KUKA KRL program: MyProgram_204().src

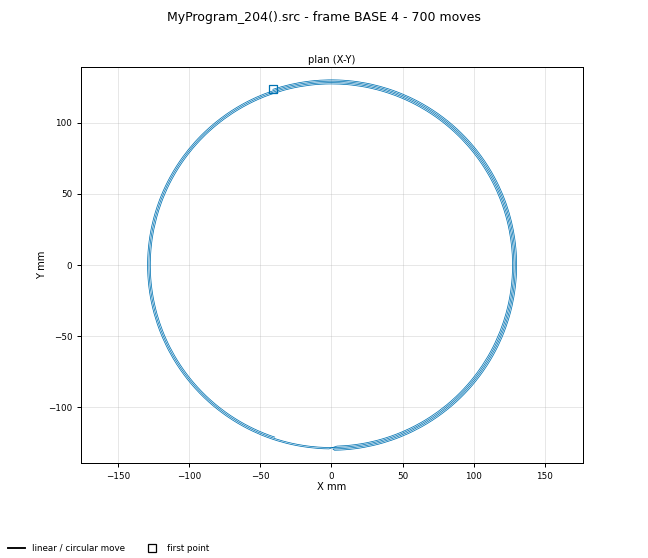
[picture p0: tool path of MyProgram_204().src in frame BASE 4, 700 of 700 moves have a stored position in this frame; points joined in program order, loops and branches not executed]
&ACCESS RVP
&REL 1
&PARAM TEMPLATE = C:\KRC\Roboter\Template\vorgabe
&PARAM EDITMASK = *
DEF MyProgram_204()
; ---- Setting reference (Base) ----
$BASE = BASE_DATA[4]

; --------------------------
; ---- Setting tool (TCP) ----
$TOOL = TOOL_DATA[3]
; --------------------------

$VEL.CP = VEL_APROX_PRINT
Startdeposition()
$VEL.CP = VEL_PRINT
LIN {X -41.1659,Y 123.6241,Z 146,A 104.1591,B 24.9489,C -1.6506,E1 24.9505,E2 342.2401} C_DIS
LIN {X -38.1321,Y 124.5933,Z 146,A 102.7568,B 24.9489,C -1.6522,E1 24.9543,E2 343.6411} C_DIS
LIN {X -35.093,Y 125.4832,Z 146,A 101.3632,B 24.9488,C -1.6536,E1 24.958,E2 345.0335} C_DIS
LIN {X -32.0884,Y 126.285,Z 146,A 100.0013,B 24.9487,C -1.6553,E1 24.9617,E2 346.3934} C_DIS
LIN {X -29.0149,Y 127.0264,Z 146,A 98.5861,B 24.9487,C -1.6553,E1 24.9655,E2 347.8103} C_DIS
LIN {X -25.7092,Y 127.7368,Z 146,A 97.1079,B 24.9485,C -1.6571,E1 24.9696,E2 349.2862} C_DIS
LIN {X -22.6845,Y 128.3085,Z 146,A 95.7157,B 24.9485,C -1.6562,E1 24.9734,E2 350.6819} C_DIS
LIN {X -19.1839,Y 128.8804,Z 146,A 94.052,B 24.9488,C -1.6522,E1 24.978,E2 352.3567} C_DIS
LIN {X -15.434,Y 129.3808,Z 146,A 92.5065,B 24.9484,C -1.6591,E1 24.9823,E2 353.887} C_DIS
LIN {X -12.0776,Y 129.7378,Z 146,A 90.8925,B 24.9488,C -1.6534,E1 24.9868,E2 355.5153} C_DIS
LIN {X -8.0122,Y 130.0517,Z 146,A 89.2662,B 24.9482,C -1.6624,E1 24.9913,E2 357.1208} C_DIS
LIN {X -5.0784,Y 130.1993,Z 146,A 87.9761,B 24.9482,C -1.6629,E1 24.9949,E2 358.4099} C_DIS
LIN {X -2.1677,Y 130.2803,Z 146,A 86.6974,B 24.9482,C -1.6634,E1 24.9984,E2 359.6878} C_DIS
LIN {X 1.1108,Y 130.2942,Z 146,A 85.0901,B 24.9486,C -1.6554,E1 25.003,E2 361.3138} C_DIS
LIN {X 5.0784,Y 130.1993,Z 146,A 83.5047,B 24.9481,C -1.6635,E1 25.0073,E2 362.8796} C_DIS
LIN {X 8.2467,Y 130.0372,Z 146,A 82.0567,B 24.9483,C -1.6609,E1 25.0114,E2 364.3334} C_DIS
LIN {X 11.7081,Y 129.7733,Z 146,A 80.4077,B 24.9487,C -1.6546,E1 25.016,E2 365.9964} C_DIS
LIN {X 15.5086,Y 129.3719,Z 146,A 78.8642,B 24.9483,C -1.6612,E1 25.0203,E2 367.5231} C_DIS
LIN {X 19.1839,Y 128.8804,Z 146,A 77.2629,B 24.9483,C -1.6622,E1 25.0247,E2 369.1206} C_DIS
LIN {X 22.1985,Y 128.3955,Z 146,A 75.9191,B 24.9483,C -1.6617,E1 25.0284,E2 370.4643} C_DIS
LIN {X 24.6619,Y 127.943,Z 146,A 74.7555,B 24.9485,C -1.6581,E1 25.0316,E2 371.635} C_DIS
LIN {X 28.256,Y 127.1998,Z 146,A 73.2021,B 24.9483,C -1.6603,E1 25.0358,E2 373.1811} C_DIS
LIN {X 31.2935,Y 126.4867,Z 146,A 71.8297,B 24.9483,C -1.6595,E1 25.0395,E2 374.5535} C_DIS
LIN {X 34.1145,Y 125.754,Z 146,A 70.5547,B 24.9484,C -1.659,E1 25.043,E2 375.8277} C_DIS
LIN {X 36.8165,Y 124.9886,Z 146,A 69.319,B 24.9484,C -1.6581,E1 25.0463,E2 377.0634} C_DIS
LIN {X 39.9416,Y 124.0254,Z 146,A 67.8799,B 24.9486,C -1.6569,E1 25.0501,E2 378.5028} C_DIS
LIN {X 42.9418,Y 123.0187,Z 146,A 66.4781,B 24.9486,C -1.6552,E1 25.0538,E2 379.906} C_DIS
LIN {X 45.9616,Y 121.9227,Z 146,A 65.0785,B 24.9487,C -1.6545,E1 25.0575,E2 381.3042} C_DIS
LIN {X 49.2138,Y 120.6475,Z 146,A 63.5495,B 24.9487,C -1.6532,E1 25.0615,E2 382.8328} C_DIS
LIN {X 52.4564,Y 119.2749,Z 146,A 61.9925,B 24.9489,C -1.651,E1 25.0655,E2 384.3913} C_DIS
LIN {X 54.9664,Y 118.1368,Z 146,A 60.7346,B 24.9492,C -1.6473,E1 25.0687,E2 385.6549} C_DIS
LIN {X 58.3801,Y 116.4901,Z 146,A 59.1188,B 24.9492,C -1.6477,E1 25.0727,E2 387.2653} C_DIS
LIN {X 61.3057,Y 114.9773,Z 146,A 57.6735,B 24.9492,C -1.6459,E1 25.0763,E2 388.7109} C_DIS
LIN {X 64.563,Y 113.1796,Z 146,A 55.9762,B 24.9496,C -1.6404,E1 25.0804,E2 390.4162} C_DIS
LIN {X 68.0397,Y 111.1243,Z 146,A 54.1884,B 24.9498,C -1.6371,E1 25.0847,E2 392.2062} C_DIS
LIN {X 71.5157,Y 108.9199,Z 146,A 52.38,B 24.95,C -1.6342,E1 25.089,E2 394.0155} C_DIS
LIN {X 74.9755,Y 106.5679,Z 146,A 50.5309,B 24.9502,C -1.6306,E1 25.0932,E2 395.8669} C_DIS
LIN {X 78.6774,Y 103.8649,Z 146,A 48.5505,B 24.9502,C -1.6288,E1 25.0977,E2 397.8444} C_DIS
LIN {X 82.0877,Y 101.1916,Z 146,A 46.6185,B 24.9506,C -1.6238,E1 25.1019,E2 399.7811} C_DIS
LIN {X 85.3172,Y 98.4841,Z 146,A 44.7731,B 24.9508,C -1.6205,E1 25.1058,E2 401.627} C_DIS
LIN {X 88.4903,Y 95.6433,Z 146,A 42.9136,B 24.951,C -1.6173,E1 25.1096,E2 403.4866} C_DIS
LIN {X 91.5168,Y 92.7515,Z 146,A 41.0777,B 24.9512,C -1.6136,E1 25.1133,E2 405.3235} C_DIS
LIN {X 94.4902,Y 89.7205,Z 146,A 39.2228,B 24.9514,C -1.61,E1 25.1169,E2 407.1788} C_DIS
LIN {X 97.316,Y 86.6472,Z 146,A 37.3918,B 24.9517,C -1.6061,E1 25.1204,E2 409.011} C_DIS
LIN {X 100.0901,Y 83.4275,Z 146,A 35.5724,B 24.9517,C -1.6042,E1 25.1236,E2 410.8265} C_DIS
LIN {X 102.7296,Y 80.155,Z 146,A 33.6589,B 24.9523,C -1.5962,E1 25.127,E2 412.7498} C_DIS
LIN {X 105.3588,Y 76.6654,Z 146,A 31.7669,B 24.9525,C -1.5929,E1 25.1301,E2 414.6406} C_DIS
LIN {X 107.8878,Y 73.0632,Z 146,A 29.8878,B 24.9525,C -1.5909,E1 25.1331,E2 416.5153} C_DIS
LIN {X 110.3417,Y 69.3023,Z 146,A 27.9203,B 24.9529,C -1.586,E1 25.1361,E2 418.4845} C_DIS
LIN {X 112.5292,Y 65.691,Z 146,A 26.0522,B 24.9532,C -1.5803,E1 25.1387,E2 420.3563} C_DIS
LIN {X 114.5867,Y 62.0329,Z 146,A 24.2001,B 24.9535,C -1.5748,E1 25.1412,E2 422.2118} C_DIS
LIN {X 116.3208,Y 58.7126,Z 146,A 22.6908,B 24.9534,C -1.5775,E1 25.1431,E2 423.7067} C_DIS
LIN {X 117.7272,Y 55.8387,Z 146,A 21.2514,B 24.9537,C -1.5717,E1 25.1449,E2 425.152} C_DIS
LIN {X 119.2263,Y 52.5651,Z 146,A 19.7299,B 24.9537,C -1.5704,E1 25.1466,E2 426.6685} C_DIS
LIN {X 120.3634,Y 49.9027,Z 146,A 18.4123,B 24.9542,C -1.5642,E1 25.1481,E2 427.9932} C_DIS
LIN {X 122.0195,Y 45.703,Z 146,A 16.484,B 24.9543,C -1.5613,E1 25.15,E2 429.9177} C_DIS
LIN {X 123.1093,Y 42.6806,Z 146,A 15.0884,B 24.9545,C -1.5579,E1 25.1513,E2 431.3134} C_DIS
LIN {X 124.1186,Y 39.6499,Z 146,A 13.6882,B 24.9548,C -1.5539,E1 25.1525,E2 432.7153} C_DIS
LIN {X 125.0483,Y 36.6127,Z 146,A 12.3025,B 24.955,C -1.5501,E1 25.1536,E2 434.1019} C_DIS
LIN {X 125.8983,Y 33.5736,Z 146,A 10.9352,B 24.9552,C -1.5469,E1 25.1546,E2 435.469} C_DIS
LIN {X 126.6698,Y 30.5342,Z 146,A 9.5775,B 24.9554,C -1.5437,E1 25.1556,E2 436.8265} C_DIS
LIN {X 127.3635,Y 27.4977,Z 146,A 8.2079,B 24.9556,C -1.5393,E1 25.1564,E2 438.1984} C_DIS
LIN {X 127.9803,Y 24.4669,Z 146,A 6.8509,B 24.9558,C -1.5351,E1 25.1571,E2 439.5573} C_DIS
LIN {X 128.5213,Y 21.4444,Z 146,A 5.5184,B 24.956,C -1.5317,E1 25.1578,E2 440.89} C_DIS
LIN {X 128.9877,Y 18.4327,Z 146,A 4.1834,B 24.9563,C -1.5277,E1 25.1583,E2 442.2266} C_DIS
LIN {X 129.3808,Y 15.434,Z 146,A 2.8295,B 24.9566,C -1.5221,E1 25.1588,E2 443.5858} C_DIS
LIN {X 129.7733,Y 11.7081,Z 146,A 1.2309,B 24.9568,C -1.5193,E1 25.1592,E2 445.1815} C_DIS
LIN {X 130.0063,Y 8.7481,Z 146,A -0.212,B 24.9574,C -1.5076,E1 25.1595,E2 446.6433} C_DIS
LIN {X 130.1993,Y 5.0784,Z 146,A -1.6641,B 24.9572,C -1.5112,E1 25.1597,E2 448.0784} C_DIS
LIN {X 130.2826,Y 2.0274,Z 146,A -3.0504,B 24.9576,C -1.5043,E1 25.1597,E2 449.4725} C_DIS
LIN {X 130.2851,Y -1.8813,Z 146,A -4.7567,B 24.9579,C -1.4993,E1 25.1597,E2 451.1805} C_DIS
LIN {X 130.1904,Y -5.305,Z 146,A -6.2523,B 24.9581,C -1.4949,E1 25.1597,E2 452.6777} C_DIS
LIN {X 130.0063,Y -8.7481,Z 146,A -7.71,B 24.9582,C -1.493,E1 25.1594,E2 454.1311} C_DIS
LIN {X 129.7229,Y -12.2325,Z 146,A -9.2888,B 24.9586,C -1.4857,E1 25.159,E2 455.7178} C_DIS
LIN {X 129.3524,Y -15.6724,Z 146,A -10.7575,B 24.9588,C -1.4835,E1 25.1585,E2 457.1829} C_DIS
LIN {X 128.8804,Y -19.1839,Z 146,A -12.3029,B 24.959,C -1.479,E1 25.1579,E2 458.7298} C_DIS
LIN {X 128.301,Y -22.7268,Z 146,A -13.9039,B 24.9594,C -1.4727,E1 25.1572,E2 460.3365} C_DIS
LIN {X 127.6814,Y -25.9814,Z 146,A -15.323,B 24.9595,C -1.4699,E1 25.1564,E2 461.7538} C_DIS
LIN {X 127.0264,Y -29.0149,Z 146,A -16.6968,B 24.9598,C -1.465,E1 25.1556,E2 463.1313} C_DIS
LIN {X 126.2312,Y -32.3004,Z 146,A -18.1777,B 24.96,C -1.4604,E1 25.1546,E2 464.6143} C_DIS
LIN {X 125.3725,Y -35.489,Z 146,A -19.6315,B 24.9603,C -1.4556,E1 25.1535,E2 466.071} C_DIS
LIN {X 124.4556,Y -38.5819,Z 146,A -21.0351,B 24.9605,C -1.4518,E1 25.1524,E2 467.4756} C_DIS
LIN {X 123.4403,Y -41.7177,Z 146,A -22.4398,B 24.9606,C -1.4496,E1 25.1511,E2 468.8776} C_DIS
LIN {X 122.5066,Y -44.3814,Z 146,A -23.7072,B 24.9609,C -1.4442,E1 25.1499,E2 470.1505} C_DIS
LIN {X 121.2828,Y -47.6258,Z 146,A -25.1893,B 24.9611,C -1.4417,E1 25.1485,E2 471.6303} C_DIS
LIN {X 120.0731,Y -50.5978,Z 146,A -26.6249,B 24.9614,C -1.436,E1 25.1469,E2 473.0716} C_DIS
LIN {X 118.7918,Y -53.5364,Z 146,A -28.0489,B 24.9617,C -1.4308,E1 25.1453,E2 474.5} C_DIS
LIN {X 117.472,Y -56.3728,Z 146,A -29.3837,B 24.9617,C -1.4288,E1 25.1437,E2 475.8324} C_DIS
LIN {X 115.9248,Y -59.4905,Z 146,A -31.0338,B 24.9624,C -1.4177,E1 25.1416,E2 477.4999} C_DIS
LIN {X 113.7905,Y -63.4816,Z 146,A -33.0095,B 24.9626,C -1.4124,E1 25.139,E2 479.4776} C_DIS
LIN {X 111.5808,Y -67.2886,Z 146,A -34.8948,B 24.9628,C -1.4094,E1 25.1363,E2 481.3603} C_DIS
LIN {X 109.288,Y -70.9517,Z 146,A -36.7607,B 24.963,C -1.4057,E1 25.1335,E2 483.2254} C_DIS
LIN {X 106.9636,Y -74.4097,Z 146,A -38.5852,B 24.9632,C -1.4009,E1 25.1306,E2 485.0524} C_DIS
LIN {X 104.5125,Y -77.8148,Z 146,A -40.4188,B 24.9635,C -1.3964,E1 25.1276,E2 486.8879} C_DIS
LIN {X 101.9488,Y -81.1445,Z 146,A -42.2562,B 24.9637,C -1.3918,E1 25.1244,E2 488.7273} C_DIS
LIN {X 99.2765,Y -84.393,Z 146,A -44.096,B 24.9639,C -1.3874,E1 25.1211,E2 490.5691} C_DIS
LIN {X 96.6485,Y -87.3906,Z 146,A -45.8895,B 24.9643,C -1.3807,E1 25.1178,E2 492.3705} C_DIS
LIN {X 93.6143,Y -90.6331,Z 146,A -47.775,B 24.9643,C -1.3793,E1 25.1142,E2 494.2511} C_DIS
LIN {X 90.6331,Y -93.6143,Z 146,A -49.6264,B 24.9646,C -1.3748,E1 25.1105,E2 496.1052} C_DIS
LIN {X 87.606,Y -96.453,Z 146,A -51.4433,B 24.9648,C -1.3708,E1 25.1067,E2 497.9241} C_DIS
LIN {X 84.5251,Y -99.1642,Z 146,A -53.2748,B 24.9651,C -1.3652,E1 25.1029,E2 499.7618} C_DIS
LIN {X 81.1445,Y -101.9488,Z 146,A -55.1532,B 24.9651,C -1.3633,E1 25.0988,E2 501.6374} C_DIS
LIN {X 77.8179,Y -104.5102,Z 146,A -56.9762,B 24.9653,C -1.3605,E1 25.0947,E2 503.4603} C_DIS
LIN {X 74.5281,Y -106.8812,Z 146,A -58.7931,B 24.9656,C -1.355,E1 25.0906,E2 505.284} C_DIS
LIN {X 70.9517,Y -109.288,Z 146,A -60.6507,B 24.9657,C -1.3532,E1 25.0863,E2 507.1397} C_DIS
LIN {X 67.1938,Y -111.6381,Z 146,A -62.622,B 24.966,C -1.3483,E1 25.0816,E2 509.1164} C_DIS
LIN {X 63.4816,Y -113.7905,Z 146,A -64.4818,B 24.966,C -1.3462,E1 25.0771,E2 510.9755} C_DIS
LIN {X 59.8462,Y -115.7437,Z 146,A -66.2101,B 24.966,C -1.3476,E1 25.0728,E2 512.6957} C_DIS
LIN {X 57.3676,Y -116.9896,Z 146,A -67.4374,B 24.9661,C -1.3452,E1 25.0697,E2 513.9254} C_DIS
LIN {X 53.9453,Y -118.6089,Z 146,A -69.0822,B 24.9661,C -1.3435,E1 25.0656,E2 515.5699} C_DIS
LIN {X 51.2764,Y -119.7851,Z 146,A -70.3402,B 24.9662,C -1.3429,E1 25.0623,E2 516.8264} C_DIS
LIN {X 48.2339,Y -121.0425,Z 146,A -71.7953,B 24.9663,C -1.3404,E1 25.0586,E2 518.2841} C_DIS
LIN {X 45.3511,Y -122.1513,Z 146,A -73.1766,B 24.9665,C -1.3373,E1 25.055,E2 519.6697} C_DIS
LIN {X 42.2564,Y -123.2564,Z 146,A -74.5919,B 24.9665,C -1.337,E1 25.0512,E2 521.083} C_DIS
LIN {X 39.2006,Y -124.2621,Z 146,A -76.023,B 24.9667,C -1.3343,E1 25.0474,E2 522.5176} C_DIS
LIN {X 36.3649,Y -125.1208,Z 146,A -77.3394,B 24.9667,C -1.3321,E1 25.0439,E2 523.8369} C_DIS
LIN {X 32.9264,Y -126.0709,Z 146,A -78.9998,B 24.9671,C -1.3257,E1 25.0394,E2 525.5101} C_DIS
LIN {X 29.1313,Y -126.9998,Z 146,A -80.599,B 24.9669,C -1.3301,E1 25.0351,E2 527.0963} C_DIS
LIN {X 25.9814,Y -127.6814,Z 146,A -81.9862,B 24.9669,C -1.3304,E1 25.0313,E2 528.4812} C_DIS
LIN {X 22.9743,Y -128.2567,Z 146,A -83.332,B 24.9669,C -1.3293,E1 25.0276,E2 529.8281} C_DIS
LIN {X 19.937,Y -128.7638,Z 146,A -84.7073,B 24.967,C -1.3272,E1 25.0238,E2 531.2071} C_DIS
LIN {X 16.5645,Y -129.2415,Z 146,A -86.2017,B 24.967,C -1.3263,E1 25.0196,E2 532.7022} C_DIS
LIN {X 13.1951,Y -129.6305,Z 146,A -87.658,B 24.967,C -1.3272,E1 25.0156,E2 534.1554} C_DIS
LIN {X 9.6067,Y -129.9437,Z 146,A -89.2621,B 24.967,C -1.3254,E1 25.0111,E2 535.7628} C_DIS
LIN {X 6.2428,Y -130.149,Z 146,A -90.8764,B 24.9675,C -1.3181,E1 25.0066,E2 537.394} C_DIS
LIN {X 2.1677,Y -130.2803,Z 146,A -92.503,B 24.9671,C -1.326,E1 25.0021,E2 539.0016} C_DIS
LIN {X 2.1677,Y -130.2803,Z 146,A -92.503,B 24.9671,C -1.326,E1 25.0021,E2 539.0016} C_DIS
Enddeposition()
LIN {X 0.9239,Y -129.3368,Z 146,A -93.0172,B 24.1837,C -1.1824,E1 24.2108,E2 539.7577} C_DIS
Startdeposition()
$VEL.CP = VEL_PRINT
LIN {X 4.2044,Y -129.2745,Z 146,A -90.6178,B 24.1815,C -1.2293,E1 24.2178,E2 537.2441} C_DIS
LIN {X 8.0458,Y -129.0909,Z 146,A -88.9904,B 24.1816,C -1.2262,E1 24.2223,E2 535.6249} C_DIS
LIN {X 12.9463,Y -128.693,Z 146,A -86.7775,B 24.1815,C -1.2291,E1 24.2285,E2 533.4063} C_DIS
LIN {X 16.7077,Y -128.2576,Z 146,A -84.5287,B 24.18,C -1.2589,E1 24.2349,E2 531.0866} C_DIS
LIN {X 21.7471,Y -127.5007,Z 146,A -83.0315,B 24.1818,C -1.2223,E1 24.2388,E2 529.6803} C_DIS
LIN {X 24.389,Y -127.0209,Z 146,A -81.7505,B 24.1815,C -1.2279,E1 24.2423,E2 528.3873} C_DIS
LIN {X 27.9389,Y -126.2892,Z 146,A -80.0921,B 24.1813,C -1.232,E1 24.2469,E2 526.7211} C_DIS
LIN {X 31.6964,Y -125.3972,Z 146,A -78.4252,B 24.1813,C -1.2315,E1 24.2514,E2 525.0579} C_DIS
LIN {X 35.0406,Y -124.5042,Z 146,A -76.8855,B 24.1813,C -1.2335,E1 24.2555,E2 523.5159} C_DIS
LIN {X 39.6598,Y -123.1109,Z 146,A -74.8628,B 24.1814,C -1.2302,E1 24.2609,E2 521.505} C_DIS
LIN {X 42.3734,Y -122.203,Z 146,A -73.4996,B 24.1811,C -1.2366,E1 24.2645,E2 520.1288} C_DIS
LIN {X 45.6538,Y -121.0161,Z 146,A -71.9964,B 24.1811,C -1.2366,E1 24.2685,E2 518.6291} C_DIS
LIN {X 48.6388,Y -119.8475,Z 146,A -70.5355,B 24.1809,C -1.2407,E1 24.2723,E2 517.1616} C_DIS
LIN {X 53.521,Y -117.7505,Z 146,A -68.2298,B 24.1809,C -1.2418,E1 24.2782,E2 514.8591} C_DIS
LIN {X 56.6438,Y -116.2796,Z 146,A -66.5962,B 24.1805,C -1.2496,E1 24.2823,E2 513.2109} C_DIS
LIN {X 64.9061,Y -111.8783,Z 146,A -62.4943,B 24.1802,C -1.2545,E1 24.2924,E2 509.1093} C_DIS
LIN {X 70.1129,Y -108.6914,Z 146,A -59.8427,B 24.1802,C -1.2569,E1 24.2987,E2 506.4605} C_DIS
LIN {X 73.18,Y -106.65,Z 146,A -58.1557,B 24.1798,C -1.2631,E1 24.3026,E2 504.7644} C_DIS
LIN {X 76.8503,Y -104.037,Z 146,A -56.1353,B 24.1796,C -1.2685,E1 24.3072,E2 502.7382} C_DIS
LIN {X 80.3501,Y -101.3581,Z 146,A -54.1965,B 24.1794,C -1.2721,E1 24.3114,E2 500.7982} C_DIS
LIN {X 83.8862,Y -98.4513,Z 146,A -52.2016,B 24.1792,C -1.275,E1 24.3157,E2 498.8041} C_DIS
LIN {X 87.2035,Y -95.5261,Z 146,A -49.7022,B 24.1776,C -1.3078,E1 24.321,E2 496.2355} C_DIS
LIN {X 90.7593,Y -92.1532,Z 146,A -48.3526,B 24.1795,C -1.2703,E1 24.3235,E2 494.9828} C_DIS
LIN {X 92.8609,Y -90.0356,Z 146,A -46.81,B 24.1787,C -1.285,E1 24.3266,E2 493.4112} C_DIS
LIN {X 95.6119,Y -87.109,Z 146,A -44.9804,B 24.1784,C -1.2922,E1 24.3301,E2 491.5726} C_DIS
LIN {X 98.4763,Y -83.8568,Z 146,A -43.0739,B 24.1782,C -1.2965,E1 24.3336,E2 489.6645} C_DIS
LIN {X 101.4916,Y -80.1818,Z 146,A -41.0186,B 24.178,C -1.2996,E1 24.3372,E2 487.6117} C_DIS
LIN {X 104.0224,Y -76.8701,Z 146,A -39.1282,B 24.1776,C -1.3069,E1 24.3403,E2 485.7128} C_DIS
LIN {X 106.9996,Y -72.6683,Z 146,A -36.1292,B 24.1753,C -1.3512,E1 24.3452,E2 482.6216} C_DIS
LIN {X 110.2998,Y -67.5537,Z 146,A -34.2932,B 24.1773,C -1.3136,E1 24.3478,E2 480.8865} C_DIS
LIN {X 112.8544,Y -63.1939,Z 146,A -32.051,B 24.1769,C -1.3204,E1 24.3509,E2 478.6399} C_DIS
LIN {X 114.62,Y -59.9279,Z 146,A -30.468,B 24.1769,C -1.3221,E1 24.353,E2 477.0613} C_DIS
LIN {X 116.1533,Y -56.8998,Z 146,A -28.9363,B 24.1765,C -1.3281,E1 24.3549,E2 475.5235} C_DIS
LIN {X 118.4291,Y -52.0014,Z 146,A -26.6306,B 24.1765,C -1.3309,E1 24.3576,E2 473.2241} C_DIS
LIN {X 119.4601,Y -49.5826,Z 146,A -25.4584,B 24.1762,C -1.3349,E1 24.3588,E2 472.0488} C_DIS
LIN {X 120.616,Y -46.6999,Z 146,A -24.0694,B 24.1759,C -1.3399,E1 24.3603,E2 470.6557} C_DIS
LIN {X 121.8745,Y -43.3132,Z 146,A -22.1514,B 24.1748,C -1.3617,E1 24.3621,E2 468.696} C_DIS
LIN {X 122.971,Y -40.0975,Z 146,A -21.0036,B 24.1755,C -1.3476,E1 24.3631,E2 467.5891} C_DIS
LIN {X 124.0699,Y -36.5487,Z 146,A -19.4234,B 24.1755,C -1.3495,E1 24.3644,E2 466.0136} C_DIS
LIN {X 124.9718,Y -33.3341,Z 146,A -17.8718,B 24.175,C -1.358,E1 24.3655,E2 464.4505} C_DIS
LIN {X 125.8855,Y -29.7043,Z 146,A -16.1834,B 24.1746,C -1.365,E1 24.3666,E2 462.7554} C_DIS
LIN {X 126.7224,Y -25.8954,Z 146,A -14.5182,B 24.1745,C -1.3673,E1 24.3676,E2 461.0945} C_DIS
LIN {X 127.3956,Y -22.3539,Z 146,A -12.8758,B 24.1741,C -1.3749,E1 24.3684,E2 459.4437} C_DIS
LIN {X 128.2631,Y -16.6661,Z 146,A -9.9027,B 24.1724,C -1.4057,E1 24.3696,E2 456.4141} C_DIS
LIN {X 128.7367,Y -12.4917,Z 146,A -8.6813,B 24.1739,C -1.378,E1 24.3699,E2 455.2673} C_DIS
LIN {X 129.1577,Y -6.9019,Z 146,A -5.9341,B 24.1727,C -1.4,E1 24.3705,E2 452.4836} C_DIS
LIN {X 129.3221,Y -2.2358,Z 146,A -4.0351,B 24.1729,C -1.3979,E1 24.3705,E2 450.6016} C_DIS
LIN {X 129.3232,Y 2.17,Z 146,A -1.5858,B 24.1711,C -1.4305,E1 24.3705,E2 448.0881} C_DIS
LIN {X 129.1818,Y 6.4224,Z 146,A -0.2608,B 24.1723,C -1.4071,E1 24.3704,E2 446.8281} C_DIS
LIN {X 128.8041,Y 11.7869,Z 146,A 2.2966,B 24.1714,C -1.424,E1 24.3698,E2 444.2454} C_DIS
LIN {X 128.3691,Y 15.837,Z 146,A 4.6153,B 24.1696,C -1.457,E1 24.369,E2 441.8609} C_DIS
LIN {X 127.6433,Y 20.8922,Z 146,A 6.1983,B 24.1712,C -1.4284,E1 24.3683,E2 440.3569} C_DIS
LIN {X 126.9954,Y 24.5227,Z 146,A 7.8199,B 24.1709,C -1.433,E1 24.3675,E2 438.734} C_DIS
LIN {X 126.1682,Y 28.4747,Z 146,A 9.6145,B 24.1706,C -1.4389,E1 24.3664,E2 436.9358} C_DIS
LIN {X 125.37,Y 31.8035,Z 146,A 11.0633,B 24.1706,C -1.4401,E1 24.3655,E2 435.4927} C_DIS
LIN {X 124.5497,Y 34.8778,Z 146,A 12.4941,B 24.1702,C -1.4456,E1 24.3644,E2 434.0571} C_DIS
LIN {X 123.4683,Y 38.5381,Z 146,A 14.3531,B 24.1694,C -1.4596,E1 24.3629,E2 432.1753} C_DIS
LIN {X 122.19,Y 42.4108,Z 146,A 15.9591,B 24.1697,C -1.4546,E1 24.3615,E2 430.5906} C_DIS
LIN {X 121.0601,Y 45.5363,Z 146,A 17.4246,B 24.1695,C -1.4587,E1 24.36,E2 429.1237} C_DIS
LIN {X 119.9067,Y 48.4921,Z 146,A 18.8661,B 24.1691,C -1.4647,E1 24.3585,E2 427.6758} C_DIS
LIN {X 118.1026,Y 52.7336,Z 146,A 20.8906,B 24.1688,C -1.4698,E1 24.3563,E2 425.6506} C_DIS
LIN {X 116.6258,Y 55.9241,Z 146,A 22.3968,B 24.1688,C -1.4716,E1 24.3545,E2 424.1484} C_DIS
LIN {X 115.0671,Y 59.066,Z 146,A 23.947,B 24.1685,C -1.4758,E1 24.3525,E2 422.5965} C_DIS
LIN {X 113.2636,Y 62.4577,Z 146,A 25.7619,B 24.1679,C -1.4864,E1 24.3501,E2 420.7658} C_DIS
LIN {X 111.3295,Y 65.8441,Z 146,A 27.4692,B 24.1677,C -1.49,E1 24.3477,E2 419.0587} C_DIS
LIN {X 108.9731,Y 69.6736,Z 146,A 29.2932,B 24.1679,C -1.4867,E1 24.345,E2 417.2524} C_DIS
LIN {X 106.8718,Y 72.8569,Z 146,A 31.0848,B 24.1673,C -1.4963,E1 24.3422,E2 415.4466} C_DIS
LIN {X 104.4728,Y 76.257,Z 146,A 32.9722,B 24.1669,C -1.5033,E1 24.3391,E2 413.5517} C_DIS
LIN {X 101.074,Y 80.7071,Z 146,A 35.1506,B 24.1675,C -1.4939,E1 24.3355,E2 411.4069} C_DIS
LIN {X 99.1815,Y 83.0217,Z 146,A 36.7336,B 24.1665,C -1.5103,E1 24.3326,E2 409.7916} C_DIS
LIN {X 96.1606,Y 86.5029,Z 146,A 39.5696,B 24.1638,C -1.556,E1 24.3271,E2 406.8575} C_DIS
LIN {X 91.85,Y 91.0667,Z 146,A 41.4539,B 24.1662,C -1.5159,E1 24.3237,E2 405.079} C_DIS
LIN {X 88.7788,Y 94.0631,Z 146,A 43.4094,B 24.1658,C -1.5228,E1 24.3197,E2 403.1153} C_DIS
LIN {X 85.4833,Y 97.0681,Z 146,A 45.3703,B 24.1656,C -1.526,E1 24.3156,E2 401.1546} C_DIS
LIN {X 81.609,Y 100.3473,Z 146,A 47.3329,B 24.1662,C -1.5159,E1 24.3115,E2 399.2244} C_DIS
LIN {X 78.0777,Y 103.1186,Z 146,A 49.6182,B 24.1651,C -1.5346,E1 24.3064,E2 396.9024} C_DIS
LIN {X 74.4187,Y 105.7896,Z 146,A 51.5752,B 24.165,C -1.5356,E1 24.3019,E2 394.9502} C_DIS
LIN {X 70.9411,Y 108.1525,Z 146,A 53.4624,B 24.1647,C -1.5399,E1 24.2975,E2 393.059} C_DIS
LIN {X 67.0886,Y 110.5834,Z 146,A 55.4658,B 24.1646,C -1.5423,E1 24.2928,E2 391.0562} C_DIS
LIN {X 63.4058,Y 112.7353,Z 146,A 57.3529,B 24.1644,C -1.545,E1 24.2882,E2 389.1685} C_DIS
LIN {X 59.5391,Y 114.8242,Z 146,A 59.1768,B 24.1646,C -1.5415,E1 24.2837,E2 387.3585} C_DIS
LIN {X 56.593,Y 116.3047,Z 146,A 60.7468,B 24.1642,C -1.5488,E1 24.2798,E2 385.7751} C_DIS
LIN {X 53.0349,Y 117.9679,Z 146,A 62.4099,B 24.1643,C -1.5471,E1 24.2756,E2 384.1205} C_DIS
LIN {X 49.5936,Y 119.4555,Z 146,A 64.0262,B 24.1643,C -1.5467,E1 24.2714,E2 382.5092} C_DIS
LIN {X 46.6078,Y 120.6518,Z 146,A 65.4667,B 24.1642,C -1.5489,E1 24.2677,E2 381.0665} C_DIS
LIN {X 43.0618,Y 121.9643,Z 146,A 67.2656,B 24.1637,C -1.5566,E1 24.2629,E2 379.2528} C_DIS
LIN {X 39.0091,Y 123.3188,Z 146,A 69.018,B 24.1641,C -1.5512,E1 24.2583,E2 377.5168} C_DIS
LIN {X 35.3983,Y 124.4042,Z 146,A 70.7735,B 24.1637,C -1.5567,E1 24.2536,E2 375.7512} C_DIS
LIN {X 31.7622,Y 125.3805,Z 146,A 72.3687,B 24.1639,C -1.5542,E1 24.2493,E2 374.1647} C_DIS
LIN {X 28.7121,Y 126.114,Z 146,A 73.7517,B 24.1639,C -1.5546,E1 24.2455,E2 372.7825} C_DIS
LIN {X 25.5775,Y 126.7871,Z 146,A 75.1911,B 24.1638,C -1.5562,E1 24.2416,E2 371.3411} C_DIS
LIN {X 21.5757,Y 127.5293,Z 146,A 77.3254,B 24.1627,C -1.5732,E1 24.2356,E2 369.1679} C_DIS
LIN {X 18.1742,Y 128.058,Z 146,A 78.9804,B 24.1623,C -1.58,E1 24.231,E2 367.4977} C_DIS
LIN {X 14.0715,Y 128.5737,Z 146,A 80.3449,B 24.1637,C -1.5574,E1 24.2274,E2 366.1893} C_DIS
LIN {X 9.1632,Y 129.0166,Z 146,A 82.4892,B 24.1637,C -1.5557,E1 24.2214,E2 364.0503} C_DIS
LIN {X 6.1891,Y 129.1935,Z 146,A 84.2824,B 24.1624,C -1.5787,E1 24.2163,E2 362.2016} C_DIS
LIN {X 2.2488,Y 129.3219,Z 146,A 85.5423,B 24.1638,C -1.5549,E1 24.2129,E2 361.0002} C_DIS
LIN {X -1.1826,Y 129.3368,Z 146,A 87.6507,B 24.1621,C -1.5831,E1 24.2068,E2 358.8229} C_DIS
LIN {X -5.6719,Y 129.2183,Z 146,A 89.0697,B 24.1638,C -1.5548,E1 24.2031,E2 357.4726} C_DIS
LIN {X -10.4326,Y 128.9207,Z 146,A 91.3757,B 24.1633,C -1.5632,E1 24.1966,E2 355.1452} C_DIS
LIN {X -14.4334,Y 128.5348,Z 146,A 93.4781,B 24.1624,C -1.5777,E1 24.1906,E2 353.0059} C_DIS
LIN {X -18.4741,Y 128.0152,Z 146,A 94.6681,B 24.1643,C -1.5471,E1 24.1876,E2 351.8898} C_DIS
LIN {X -21.3457,Y 127.5676,Z 146,A 96.0606,B 24.1641,C -1.5512,E1 24.1837,E2 350.486} C_DIS
LIN {X -24.6883,Y 126.9637,Z 146,A 97.7247,B 24.1637,C -1.5576,E1 24.1791,E2 348.8044} C_DIS
LIN {X -28.795,Y 126.0951,Z 146,A 99.456,B 24.1641,C -1.5499,E1 24.1744,E2 347.0898} C_DIS
LIN {X -32.5621,Y 125.1775,Z 146,A 101.2988,B 24.1639,C -1.5541,E1 24.1694,E2 345.234} C_DIS
LIN {X -36.2023,Y 124.1713,Z 146,A 102.98,B 24.1639,C -1.5527,E1 24.1648,E2 343.5533} C_DIS
LIN {X -39.6345,Y 123.119,Z 146,A 104.4461,B 24.1644,C -1.545,E1 24.161,E2 342.1034} C_DIS
LIN {X -47.1522,Y 120.4402,Z 146,A 108.0019,B 24.1647,C -1.5413,E1 24.1517,E2 338.5492} C_DIS
LIN {X -52.6198,Y 118.1536,Z 146,A 110.3757,B 24.1656,C -1.5257,E1 24.1457,E2 336.2079} C_DIS
LIN {X -56.0134,Y 116.5831,Z 146,A 112.2625,B 24.1651,C -1.5339,E1 24.1408,E2 334.2962} C_DIS
LIN {X -59.0106,Y 115.0953,Z 146,A 113.8105,B 24.1651,C -1.5345,E1 24.1369,E2 332.7424} C_DIS
LIN {X -62.8395,Y 113.0522,Z 146,A 115.808,B 24.1651,C -1.5347,E1 24.132,E2 330.7385} C_DIS
LIN {X -66.6481,Y 110.8499,Z 146,A 117.7933,B 24.1651,C -1.5328,E1 24.1272,E2 328.7516} C_DIS
LIN {X -70.4343,Y 108.483,Z 146,A 120.1018,B 24.1645,C -1.5444,E1 24.1217,E2 326.4069} C_DIS
LIN {X -73.7242,Y 106.2748,Z 146,A 122.1725,B 24.1638,C -1.5556,E1 24.1169,E2 324.3014} C_DIS
LIN {X -78.1894,Y 103.0344,Z 146,A 123.7093,B 24.1666,C -1.5083,E1 24.1137,E2 322.875} C_DIS
LIN {X -81.9997,Y 100.0281,Z 146,A 126.1808,B 24.166,C -1.5184,E1 24.1083,E2 320.3692} C_DIS
LIN {X -85.5473,Y 97.0114,Z 146,A 128.212,B 24.1664,C -1.5122,E1 24.104,E2 318.3449} C_DIS
LIN {X -88.9697,Y 93.883,Z 146,A 130.5078,B 24.166,C -1.5185,E1 24.0992,E2 316.0239} C_DIS
LIN {X -91.4109,Y 91.508,Z 146,A 132.0358,B 24.1662,C -1.5157,E1 24.0962,E2 314.4961} C_DIS
LIN {X -93.8238,Y 89.0325,Z 146,A 133.0862,B 24.1677,C -1.4898,E1 24.0943,E2 313.5046} C_DIS
LIN {X -95.9392,Y 86.7483,Z 146,A 134.675,B 24.1673,C -1.4959,E1 24.0913,E2 311.8935} C_DIS
LIN {X -100.6523,Y 81.2321,Z 146,A 137.74,B 24.1682,C -1.4806,E1 24.0858,E2 308.8514} C_DIS
LIN {X -104.3902,Y 76.3694,Z 146,A 140.5807,B 24.1683,C -1.4788,E1 24.081,E2 306.001} C_DIS
LIN {X -106.7035,Y 73.1021,Z 146,A 142.417,B 24.1684,C -1.4767,E1 24.078,E2 304.1604} C_DIS
LIN {X -109.0948,Y 69.4835,Z 146,A 144.4029,B 24.1686,C -1.4742,E1 24.075,E2 302.1704} C_DIS
LIN {X -111.3739,Y 65.7684,Z 146,A 146.3566,B 24.1688,C -1.4697,E1 24.0722,E2 300.2174} C_DIS
LIN {X -113.6346,Y 61.78,Z 146,A 148.3805,B 24.1692,C -1.4634,E1 24.0695,E2 298.198} C_DIS
LIN {X -115.3403,Y 58.5294,Z 146,A 149.8692,B 24.1698,C -1.4523,E1 24.0676,E2 296.7281} C_DIS
LIN {X -116.7979,Y 55.5639,Z 146,A 151.4145,B 24.1698,C -1.4515,E1 24.0657,E2 295.176} C_DIS
LIN {X -118.3871,Y 52.0977,Z 146,A 153.1821,B 24.17,C -1.4499,E1 24.0637,E2 293.4024} C_DIS
LIN {X -120.2037,Y 47.7553,Z 146,A 155.1596,B 24.1706,C -1.4386,E1 24.0616,E2 291.4414} C_DIS
LIN {X -121.3081,Y 44.8742,Z 146,A 157.1033,B 24.1694,C -1.4605,E1 24.0597,E2 289.4323} C_DIS
LIN {X -122.7332,Y 40.8124,Z 146,A 158.1312,B 24.1719,C -1.4147,E1 24.0589,E2 288.511} C_DIS
LIN {X -123.9982,Y 36.7936,Z 146,A 160.2194,B 24.1717,C -1.4187,E1 24.0571,E2 286.4004} C_DIS
LIN {X -125.0479,Y 33.0487,Z 146,A 162.1282,B 24.1716,C -1.4216,E1 24.0556,E2 284.4731} C_DIS
LIN {X -126.3127,Y 27.8299,Z 146,A 164.5779,B 24.1718,C -1.4171,E1 24.0541,E2 282.0195} C_DIS
LIN {X -127.048,Y 24.2471,Z 146,A 166.1364,B 24.1722,C -1.4091,E1 24.0532,E2 280.4711} C_DIS
LIN {X -127.7251,Y 20.3912,Z 146,A 167.9716,B 24.1723,C -1.4079,E1 24.0524,E2 278.6274} C_DIS
LIN {X -128.2633,Y 16.6644,Z 146,A 169.6083,B 24.1727,C -1.4011,E1 24.0518,E2 276.9973} C_DIS
LIN {X -128.7404,Y 12.4535,Z 146,A 171.447,B 24.1731,C -1.3932,E1 24.0512,E2 275.1665} C_DIS
LIN {X -129.0447,Y 8.7784,Z 146,A 173.2366,B 24.1731,C -1.3949,E1 24.0509,E2 273.3617} C_DIS
LIN {X -129.258,Y 4.6588,Z 146,A 175.0395,B 24.1734,C -1.3878,E1 24.0507,E2 271.5649} C_DIS
LIN {X -129.344,Y 0.3403,Z 146,A 177.0307,B 24.1735,C -1.3851,E1 24.0507,E2 269.568} C_DIS
LIN {X -129.2872,Y -3.7469,Z 146,A 178.6919,B 24.1742,C -1.3724,E1 24.0507,E2 267.9275} C_DIS
LIN {X -129.108,Y -7.7669,Z 146,A -179.505,B 24.1745,C -1.3676,E1 24.051,E2 266.1251} C_DIS
LIN {X -128.8318,Y -11.4843,Z 146,A -177.7439,B 24.1745,C -1.3672,E1 24.0514,E2 264.3539} C_DIS
LIN {X -128.4217,Y -15.3954,Z 146,A -176.1034,B 24.175,C -1.357,E1 24.0519,E2 262.7283} C_DIS
LIN {X -127.897,Y -19.281,Z 146,A -174.2729,B 24.1751,C -1.3557,E1 24.0526,E2 260.8897} C_DIS
LIN {X -127.3069,Y -22.8493,Z 146,A -172.747,B 24.1756,C -1.3471,E1 24.0533,E2 259.3754} C_DIS
LIN {X -126.6363,Y -26.3182,Z 146,A -171.0414,B 24.1755,C -1.3485,E1 24.0543,E2 257.6559} C_DIS
LIN {X -125.7376,Y -30.3179,Z 146,A -169.3024,B 24.176,C -1.3394,E1 24.0554,E2 255.9288} C_DIS
LIN {X -124.7197,Y -34.27,Z 146,A -167.6158,B 24.1765,C -1.3282,E1 24.0566,E2 254.2594} C_DIS
LIN {X -122.5054,Y -41.4963,Z 146,A -164.1757,B 24.1769,C -1.3221,E1 24.0594,E2 250.8138} C_DIS
LIN {X -121.0764,Y -45.4929,Z 146,A -162.2494,B 24.177,C -1.3186,E1 24.0613,E2 248.8848} C_DIS
LIN {X -119.9011,Y -48.5058,Z 146,A -160.8157,B 24.1773,C -1.3144,E1 24.0628,E2 247.4531} C_DIS
LIN {X -118.6374,Y -51.5197,Z 146,A -159.3606,B 24.1775,C -1.3105,E1 24.0644,E2 245.9992} C_DIS
LIN {X -117.1428,Y -54.8361,Z 146,A -157.7669,B 24.1777,C -1.3051,E1 24.0662,E2 244.4099} C_DIS
LIN {X -115.9444,Y -57.3233,Z 146,A -156.5053,B 24.1778,C -1.3034,E1 24.0678,E2 243.1453} C_DIS
LIN {X -114.4681,Y -60.2172,Z 146,A -154.6449,B 24.177,C -1.3188,E1 24.0702,E2 241.2369} C_DIS
LIN {X -112.6183,Y -63.6138,Z 146,A -153.4938,B 24.1786,C -1.2881,E1 24.0717,E2 240.1548} C_DIS
LIN {X -111.2778,Y -65.9312,Z 146,A -152.0301,B 24.1781,C -1.2977,E1 24.0738,E2 238.6598} C_DIS
LIN {X -108.9873,Y -69.6515,Z 146,A -150.0963,B 24.1784,C -1.2925,E1 24.0767,E2 236.7285} C_DIS
LIN {X -106.291,Y -73.7008,Z 146,A -147.9068,B 24.1786,C -1.2885,E1 24.0801,E2 234.5375} C_DIS
LIN {X -103.5957,Y -77.4438,Z 146,A -145.8104,B 24.1786,C -1.2858,E1 24.0836,E2 232.437} C_DIS
LIN {X -101.3694,Y -80.336,Z 146,A -144.2213,B 24.179,C -1.2806,E1 24.0863,E2 230.8531} C_DIS
LIN {X -98.5758,Y -83.7398,Z 146,A -142.291,B 24.1792,C -1.275,E1 24.0898,E2 228.9272} C_DIS
LIN {X -95.7358,Y -86.9724,Z 146,A -140.3619,B 24.1794,C -1.2718,E1 24.0934,E2 226.9972} C_DIS
LIN {X -92.6345,Y -90.2694,Z 146,A -138.3171,B 24.1795,C -1.2692,E1 24.0973,E2 224.9496} C_DIS
LIN {X -89.5084,Y -93.3693,Z 146,A -136.4037,B 24.1798,C -1.2633,E1 24.1011,E2 223.0423} C_DIS
LIN {X -86.4063,Y -96.2471,Z 146,A -134.5001,B 24.1799,C -1.2609,E1 24.1051,E2 221.1367} C_DIS
LIN {X -82.9266,Y -99.2612,Z 146,A -132.4527,B 24.1801,C -1.2573,E1 24.1094,E2 219.0899} C_DIS
LIN {X -79.556,Y -101.983,Z 146,A -130.499,B 24.1802,C -1.2553,E1 24.1137,E2 217.1334} C_DIS
LIN {X -76.1767,Y -104.5312,Z 146,A -128.6148,B 24.1803,C -1.2525,E1 24.1179,E2 215.2493} C_DIS
LIN {X -73.4891,Y -106.4379,Z 146,A -127.1538,B 24.1805,C -1.25,E1 24.1213,E2 213.789} C_DIS
LIN {X -69.4441,Y -109.12,Z 146,A -125.0588,B 24.1808,C -1.244,E1 24.1262,E2 211.7019} C_DIS
LIN {X -65.8279,Y -111.339,Z 146,A -123.1037,B 24.1808,C -1.2448,E1 24.1309,E2 209.7386} C_DIS
LIN {X -61.7923,Y -113.6279,Z 146,A -121.0558,B 24.1808,C -1.2416,E1 24.1359,E2 207.6924} C_DIS
LIN {X -58.5285,Y -115.3407,Z 146,A -119.5222,B 24.1812,C -1.2348,E1 24.1396,E2 206.1712} C_DIS
LIN {X -55.57,Y -116.795,Z 146,A -118.0701,B 24.1813,C -1.2326,E1 24.1433,E2 204.7206} C_DIS
LIN {X -51.9399,Y -118.4557,Z 146,A -116.3749,B 24.1816,C -1.227,E1 24.1476,E2 203.0346} C_DIS
LIN {X -49.3307,Y -119.5653,Z 146,A -115.0461,B 24.1815,C -1.2292,E1 24.151,E2 201.6973} C_DIS
LIN {X -45.6878,Y -121.0034,Z 146,A -113.2603,B 24.1815,C -1.23,E1 24.1557,E2 199.9057} C_DIS
LIN {X -41.5181,Y -122.4982,Z 146,A -111.2182,B 24.1813,C -1.2321,E1 24.1611,E2 197.8543} C_DIS
LIN {X -37.9001,Y -123.6636,Z 146,A -109.659,B 24.1817,C -1.2248,E1 24.1652,E2 196.3101} C_DIS
LIN {X -34.7933,Y -124.5734,Z 146,A -108.2125,B 24.1817,C -1.2245,E1 24.1691,E2 194.8621} C_DIS
LIN {X -31.7425,Y -125.3855,Z 146,A -106.8171,B 24.1817,C -1.2235,E1 24.1729,E2 193.467} C_DIS
LIN {X -28.6195,Y -126.1352,Z 146,A -105.4235,B 24.1818,C -1.2213,E1 24.1766,E2 192.0768} C_DIS
LIN {X -25.2291,Y -126.858,Z 146,A -103.3886,B 24.1807,C -1.2451,E1 24.1824,E2 189.9814} C_DIS
LIN {X -21.3246,Y -127.5712,Z 146,A -101.8898,B 24.1813,C -1.2318,E1 24.1864,E2 188.5136} C_DIS
LIN {X -15.977,Y -128.3524,Z 146,A -99.2547,B 24.1808,C -1.2431,E1 24.1938,E2 185.8488} C_DIS
LIN {X -12.1579,Y -128.7688,Z 146,A -98.1092,B 24.1821,C -1.2155,E1 24.1968,E2 184.7699} C_DIS
LIN {X -9.2477,Y -129.0104,Z 146,A -96.4928,B 24.1814,C -1.2314,E1 24.2014,E2 183.1141} C_DIS
LIN {X -5.5534,Y -129.2231,Z 146,A -94.9846,B 24.1817,C -1.225,E1 24.2056,E2 181.6211} C_DIS
LIN {X -1.7194,Y -129.3307,Z 146,A -93.1397,B 24.1813,C -1.2325,E1 24.2108,E2 179.7577} C_DIS
LIN {X -1.7194,Y -129.3307,Z 146,A -93.1397,B 24.1813,C -1.2325,E1 24.2108,E2 179.7577} C_DIS
Enddeposition()
LIN {X 0.9203,Y -128.358,Z 146,A -92.4489,B 23.3003,C -1.0524,E1 23.3237,E2 179.3994} C_DIS
Startdeposition()
$VEL.CP = VEL_PRINT
LIN {X -4.1683,Y -128.3182,Z 146,A -95.555,B 23.3019,C -1.013,E1 23.3147,E2 182.6053} C_DIS
LIN {X -9.1773,Y -128.0561,Z 146,A -97.0508,B 23.3005,C -1.0472,E1 23.3108,E2 184.0152} C_DIS
LIN {X -14.6666,Y -127.545,Z 146,A -99.4787,B 23.3005,C -1.0489,E1 23.304,E2 186.4402} C_DIS
LIN {X -19.0574,Y -126.9627,Z 146,A -101.7416,B 23.3009,C -1.0362,E1 23.2977,E2 188.7372} C_DIS
LIN {X -23.8464,Y -126.1504,Z 146,A -103.7909,B 23.3007,C -1.0424,E1 23.2921,E2 190.773} C_DIS
LIN {X -27.9161,Y -125.3142,Z 146,A -105.694,B 23.3007,C -1.041,E1 23.2869,E2 192.6822} C_DIS
LIN {X -31.4314,Y -124.4772,Z 146,A -107.1322,B 23.3004,C -1.0499,E1 23.283,E2 194.1} C_DIS
LIN {X -34.5154,Y -123.6575,Z 146,A -108.6359,B 23.3004,C -1.0472,E1 23.2789,E2 195.6131} C_DIS
LIN {X -38.0302,Y -122.623,Z 146,A -110.3819,B 23.3006,C -1.0434,E1 23.2742,E2 197.372} C_DIS
LIN {X -41.2672,Y -121.5732,Z 146,A -112.1324,B 23.301,C -1.0341,E1 23.2695,E2 199.1495} C_DIS
LIN {X -44.4655,Y -120.4393,Z 146,A -113.371,B 23.3005,C -1.0479,E1 23.2664,E2 200.3558} C_DIS
LIN {X -47.7738,Y -119.1644,Z 146,A -114.7875,B 23.3001,C -1.057,E1 23.2627,E2 201.7526} C_DIS
LIN {X -51.813,Y -117.4661,Z 146,A -116.8847,B 23.3002,C -1.0527,E1 23.2573,E2 203.8661} C_DIS
LIN {X -55.1249,Y -115.9471,Z 146,A -118.4063,B 23.3,C -1.0593,E1 23.2535,E2 205.3749} C_DIS
LIN {X -57.9207,Y -114.5764,Z 146,A -119.8842,B 23.3,C -1.0571,E1 23.2498,E2 206.8628} C_DIS
LIN {X -61.1682,Y -112.8782,Z 146,A -121.642,B 23.3002,C -1.0537,E1 23.2454,E2 208.6343} C_DIS
LIN {X -65.2176,Y -110.5876,Z 146,A -123.7968,B 23.3002,C -1.0532,E1 23.2402,E2 210.7974} C_DIS
LIN {X -70.2943,Y -107.4326,Z 146,A -126.3988,B 23.2999,C -1.0603,E1 23.2341,E2 213.3904} C_DIS
LIN {X -73.3866,Y -105.3439,Z 146,A -128.3556,B 23.3004,C -1.0502,E1 23.2295,E2 215.3801} C_DIS
LIN {X -76.4568,Y -103.1375,Z 146,A -129.7535,B 23.2997,C -1.0659,E1 23.2264,E2 216.7435} C_DIS
LIN {X -80.0167,Y -100.4005,Z 146,A -131.8244,B 23.2997,C -1.0666,E1 23.2219,E2 218.8207} C_DIS
LIN {X -83.611,Y -97.4278,Z 146,A -133.8441,B 23.2994,C -1.0733,E1 23.2176,E2 220.8319} C_DIS
LIN {X -86.9341,Y -94.4742,Z 146,A -135.7933,B 23.2991,C -1.0789,E1 23.2135,E2 222.7754} C_DIS
LIN {X -90.028,Y -91.5309,Z 146,A -137.6821,B 23.2989,C -1.0836,E1 23.2098,E2 224.6607} C_DIS
LIN {X -92.9181,Y -88.5955,Z 146,A -139.5292,B 23.2988,C -1.0872,E1 23.2062,E2 226.5072} C_DIS
LIN {X -95.8255,Y -85.4428,Z 146,A -141.5089,B 23.2987,C -1.0887,E1 23.2024,E2 228.4927} C_DIS
LIN {X -98.6705,Y -82.141,Z 146,A -143.5049,B 23.2986,C -1.091,E1 23.1988,E2 230.4927} C_DIS
LIN {X -100.963,Y -79.3057,Z 146,A -145.4714,B 23.2991,C -1.0802,E1 23.1954,E2 232.4966} C_DIS
LIN {X -103.3845,Y -76.1221,Z 146,A -146.9021,B 23.2982,C -1.0999,E1 23.1931,E2 233.8846} C_DIS
LIN {X -105.7523,Y -72.797,Z 146,A -148.9007,B 23.2983,C -1.0969,E1 23.1898,E2 235.9016} C_DIS
LIN {X -108.6387,Y -68.4146,Z 146,A -151.0788,B 23.2977,C -1.1101,E1 23.1866,E2 238.0581} C_DIS
LIN {X -110.8783,Y -64.7229,Z 146,A -152.747,B 23.297,C -1.1264,E1 23.1842,E2 239.6941} C_DIS
LIN {X -112.5076,Y -61.8472,Z 146,A -154.7042,B 23.2978,C -1.1096,E1 23.1815,E2 241.705} C_DIS
LIN {X -114.9185,Y -57.2398,Z 146,A -156.7509,B 23.2969,C -1.1279,E1 23.1789,E2 243.7172} C_DIS
LIN {X -116.4628,Y -54.0266,Z 146,A -158.3995,B 23.2969,C -1.1299,E1 23.1769,E2 245.3702} C_DIS
LIN {X -118.1301,Y -50.2818,Z 146,A -160.3347,B 23.2968,C -1.1307,E1 23.1748,E2 247.3151} C_DIS
LIN {X -119.6007,Y -46.6706,Z 146,A -161.9377,B 23.2963,C -1.1417,E1 23.1731,E2 248.8999} C_DIS
LIN {X -120.8506,Y -43.3317,Z 146,A -163.5725,B 23.2962,C -1.1445,E1 23.1716,E2 250.5375} C_DIS
LIN {X -122.3617,Y -38.8602,Z 146,A -165.9293,B 23.2964,C -1.1402,E1 23.1695,E2 252.9198} C_DIS
LIN {X -123.5294,Y -34.9734,Z 146,A -167.8111,B 23.2962,C -1.1427,E1 23.168,E2 254.8071} C_DIS
LIN {X -124.3747,Y -31.8351,Z 146,A -168.9512,B 23.2954,C -1.1604,E1 23.1673,E2 255.9093} C_DIS
LIN {X -125.1688,Y -28.5528,Z 146,A -170.4829,B 23.2952,C -1.164,E1 23.1663,E2 257.4416} C_DIS
LIN {X -125.9825,Y -24.7244,Z 146,A -172.2069,B 23.2949,C -1.1704,E1 23.1653,E2 259.1603} C_DIS
LIN {X -126.6197,Y -21.2128,Z 146,A -173.8567,B 23.2949,C -1.173,E1 23.1645,E2 260.814} C_DIS
LIN {X -127.2108,Y -17.3311,Z 146,A -175.6929,B 23.2947,C -1.175,E1 23.1638,E2 262.657} C_DIS
LIN {X -127.6233,Y -13.9597,Z 146,A -177.2048,B 23.2945,C -1.18,E1 23.1633,E2 264.1659} C_DIS
LIN {X -128.023,Y -9.6301,Z 146,A -179.1065,B 23.2941,C -1.1879,E1 23.1629,E2 266.0601} C_DIS
LIN {X -128.2457,Y -5.9834,Z 146,A 179.1582,B 23.2941,C -1.1887,E1 23.1626,E2 267.8046} C_DIS
LIN {X -128.3658,Y -2.192,Z 146,A 177.5875,B 23.2936,C -1.1993,E1 23.1625,E2 269.3584} C_DIS
LIN {X -128.3634,Y 2.3327,Z 146,A 175.4994,B 23.2934,C -1.2029,E1 23.1625,E2 271.451} C_DIS
LIN {X -128.2304,Y 6.2886,Z 146,A 173.7677,B 23.293,C -1.2101,E1 23.1627,E2 273.1756} C_DIS
LIN {X -128.015,Y 9.7394,Z 146,A 172.09,B 23.293,C -1.2094,E1 23.1631,E2 274.866} C_DIS
LIN {X -127.6781,Y 13.4502,Z 146,A 170.5096,B 23.2926,C -1.2183,E1 23.1635,E2 276.4341} C_DIS
LIN {X -127.199,Y 17.4209,Z 146,A 168.6041,B 23.2926,C -1.2189,E1 23.1642,E2 278.3503} C_DIS
LIN {X -126.6275,Y 21.1655,Z 146,A 167.0157,B 23.2921,C -1.2287,E1 23.1649,E2 279.924} C_DIS
LIN {X -125.9035,Y 25.1208,Z 146,A 165.2465,B 23.2918,C -1.2356,E1 23.1658,E2 281.6871} C_DIS
LIN {X -124.2579,Y 32.2954,Z 146,A 161.8066,B 23.2916,C -1.2394,E1 23.168,E2 285.1389} C_DIS
LIN {X -123.1231,Y 36.3768,Z 146,A 159.6856,B 23.2918,C -1.2357,E1 23.1697,E2 287.2827} C_DIS
LIN {X -122.1395,Y 39.5558,Z 146,A 158.6584,B 23.2905,C -1.2597,E1 23.1705,E2 288.2552} C_DIS
LIN {X -121.2894,Y 42.0874,Z 146,A 157.239,B 23.2908,C -1.2538,E1 23.1718,E2 289.6984} C_DIS
LIN {X -119.7515,Y 46.2827,Z 146,A 155.3369,B 23.2903,C -1.2639,E1 23.1736,E2 291.5865} C_DIS
LIN {X -117.5214,Y 51.6894,Z 146,A 152.5198,B 23.2903,C -1.263,E1 23.1767,E2 294.4226} C_DIS
LIN {X -115.8628,Y 55.3014,Z 146,A 150.9438,B 23.2897,C -1.2768,E1 23.1785,E2 295.9729} C_DIS
LIN {X -114.5102,Y 58.0507,Z 146,A 149.4853,B 23.2897,C -1.277,E1 23.1804,E2 297.4394} C_DIS
LIN {X -112.9198,Y 61.0916,Z 146,A 147.8426,B 23.2897,C -1.2767,E1 23.1825,E2 299.0922} C_DIS
LIN {X -110.6659,Y 65.0845,Z 146,A 145.8032,B 23.2893,C -1.283,E1 23.1854,E2 301.1272} C_DIS
LIN {X -108.3389,Y 68.8895,Z 146,A 143.7815,B 23.2891,C -1.2873,E1 23.1884,E2 303.1491} C_DIS
LIN {X -106.1047,Y 72.2831,Z 146,A 141.9987,B 23.2888,C -1.2936,E1 23.1911,E2 304.9253} C_DIS
LIN {X -103.6675,Y 75.7369,Z 146,A 140.386,B 23.2879,C -1.3105,E1 23.1937,E2 306.5037} C_DIS
LIN {X -100.6151,Y 79.7468,Z 146,A 136.9682,B 23.2902,C -1.2669,E1 23.1998,E2 310.0499} C_DIS
LIN {X -96.5001,Y 84.6804,Z 146,A 135.2119,B 23.2873,C -1.3215,E1 23.2028,E2 311.6761} C_DIS
LIN {X -91.8797,Y 89.6724,Z 146,A 132.1958,B 23.2869,C -1.3298,E1 23.2085,E2 314.6853} C_DIS
LIN {X -88.83,Y 92.694,Z 146,A 129.9894,B 23.2873,C -1.3218,E1 23.2129,E2 316.9219} C_DIS
LIN {X -82.9843,Y 97.9621,Z 146,A 125.9607,B 23.288,C -1.3076,E1 23.2215,E2 321.0039} C_DIS
LIN {X -79.5017,Y 100.809,Z 146,A 124.4197,B 23.2867,C -1.332,E1 23.2247,E2 322.4892} C_DIS
LIN {X -76.9234,Y 102.7901,Z 146,A 122.6498,B 23.2873,C -1.3213,E1 23.2288,E2 324.2932} C_DIS
LIN {X -73.9837,Y 104.925,Z 146,A 121.3365,B 23.2864,C -1.3379,E1 23.2317,E2 325.5693} C_DIS
LIN {X -70.2545,Y 107.4588,Z 146,A 119.2594,B 23.2864,C -1.339,E1 23.2365,E2 327.651} C_DIS
LIN {X -66.42,Y 109.8695,Z 146,A 117.3455,B 23.2859,C -1.3474,E1 23.241,E2 329.5501} C_DIS
LIN {X -63.0093,Y 111.8605,Z 146,A 115.5122,B 23.2859,C -1.3474,E1 23.2455,E2 331.3891} C_DIS
LIN {X -58.9679,Y 114.0432,Z 146,A 113.4158,B 23.2859,C -1.3488,E1 23.2506,E2 333.4884} C_DIS
LIN {X -55.5613,Y 115.7386,Z 146,A 111.8753,B 23.2853,C -1.3584,E1 23.2545,E2 335.0087} C_DIS
LIN {X -51.6467,Y 117.5392,Z 146,A 109.7631,B 23.2856,C -1.353,E1 23.2599,E2 337.1403} C_DIS
LIN {X -48.1013,Y 119.0324,Z 146,A 108.0865,B 23.2854,C -1.3572,E1 23.2642,E2 338.8104} C_DIS
LIN {X -41.1811,Y 121.6018,Z 146,A 104.9586,B 23.2847,C -1.3687,E1 23.2724,E2 341.9159} C_DIS
LIN {X -36.0492,Y 123.219,Z 146,A 102.4797,B 23.2847,C -1.3679,E1 23.279,E2 344.4013} C_DIS
LIN {X -32.696,Y 124.1516,Z 146,A 100.7859,B 23.285,C -1.3633,E1 23.2836,E2 346.1097} C_DIS
LIN {X -28.7016,Y 125.1348,Z 146,A 99.0167,B 23.2848,C -1.3679,E1 23.2884,E2 347.8698} C_DIS
LIN {X -24.4091,Y 126.0428,Z 146,A 97.0839,B 23.2846,C -1.3707,E1 23.2936,E2 349.798} C_DIS
LIN {X -20.6404,Y 126.7152,Z 146,A 95.4508,B 23.2844,C -1.3753,E1 23.2981,E2 351.4212} C_DIS
LIN {X -17.7812,Y 127.1475,Z 146,A 93.9369,B 23.2849,C -1.3661,E1 23.3024,E2 352.9597} C_DIS
LIN {X -13.848,Y 127.6353,Z 146,A 92.4349,B 23.2842,C -1.3791,E1 23.3064,E2 354.4299} C_DIS
LIN {X -7.7186,Y 128.1523,Z 146,A 89.7316,B 23.284,C -1.3821,E1 23.314,E2 357.1267} C_DIS
LIN {X -1.2386,Y 128.3796,Z 146,A 86.8237,B 23.284,C -1.3822,E1 23.3221,E2 360.0348} C_DIS
LIN {X 5.3995,Y 128.2714,Z 146,A 83.9915,B 23.2836,C -1.3885,E1 23.3299,E2 362.8508} C_DIS
LIN {X 10.6849,Y 127.939,Z 146,A 81.413,B 23.2842,C -1.3785,E1 23.3372,E2 365.4532} C_DIS
LIN {X 13.4904,Y 127.6738,Z 146,A 79.7143,B 23.2853,C -1.3582,E1 23.342,E2 367.202} C_DIS
LIN {X 17.1753,Y 127.2309,Z 146,A 78.5006,B 23.2842,C -1.378,E1 23.3453,E2 368.3646} C_DIS
LIN {X 20.4714,Y 126.7434,Z 146,A 76.9909,B 23.2843,C -1.3765,E1 23.3494,E2 369.8766} C_DIS
LIN {X 23.6099,Y 126.1956,Z 146,A 75.6114,B 23.2843,C -1.3779,E1 23.3532,E2 371.251} C_DIS
LIN {X 26.8887,Y 125.537,Z 146,A 74.0847,B 23.2843,C -1.3756,E1 23.3574,E2 372.7813} C_DIS
LIN {X 29.7822,Y 124.8824,Z 146,A 72.6847,B 23.2846,C -1.3713,E1 23.3612,E2 374.19} C_DIS
LIN {X 33.2882,Y 123.9936,Z 146,A 71.0956,B 23.2846,C -1.3715,E1 23.3655,E2 375.7761} C_DIS
LIN {X 37.2683,Y 122.8562,Z 146,A 69.4644,B 23.2841,C -1.3802,E1 23.3698,E2 377.3824} C_DIS
LIN {X 41.5169,Y 121.4871,Z 146,A 67.2131,B 23.2849,C -1.3664,E1 23.3759,E2 379.6638} C_DIS
LIN {X 44.8383,Y 120.2997,Z 146,A 65.7767,B 23.2846,C -1.3714,E1 23.3796,E2 381.0844} C_DIS
LIN {X 49.3665,Y 118.5133,Z 146,A 63.6441,B 23.2846,C -1.371,E1 23.3851,E2 383.2128} C_DIS
LIN {X 52.3428,Y 117.2291,Z 146,A 62.2169,B 23.2846,C -1.3703,E1 23.3888,E2 384.638} C_DIS
LIN {X 54.8314,Y 116.0873,Z 146,A 60.8176,B 23.2852,C -1.3604,E1 23.3923,E2 386.0582} C_DIS
LIN {X 58.0596,Y 114.5057,Z 146,A 59.3447,B 23.285,C -1.3646,E1 23.396,E2 387.5165} C_DIS
LIN {X 61.1891,Y 112.8669,Z 146,A 57.6662,B 23.2854,C -1.3576,E1 23.4002,E2 389.2074} C_DIS
LIN {X 65.0409,Y 110.6914,Z 146,A 55.8996,B 23.285,C -1.3645,E1 23.4044,E2 390.9507} C_DIS
LIN {X 67.8483,Y 108.9932,Z 146,A 54.2889,B 23.2855,C -1.3553,E1 23.4083,E2 392.5792} C_DIS
LIN {X 71.1765,Y 106.8495,Z 146,A 52.451,B 23.2858,C -1.3491,E1 23.4126,E2 394.4262} C_DIS
LIN {X 74.8398,Y 104.3166,Z 146,A 50.4718,B 23.286,C -1.3461,E1 23.4171,E2 396.4056} C_DIS
LIN {X 78.224,Y 101.8037,Z 146,A 48.5875,B 23.2862,C -1.3426,E1 23.4213,E2 398.2914} C_DIS
LIN {X 80.914,Y 99.6795,Z 146,A 47.0259,B 23.2864,C -1.3381,E1 23.4247,E2 399.8578} C_DIS
LIN {X 84.3224,Y 96.8125,Z 146,A 45.0982,B 23.2864,C -1.3371,E1 23.4288,E2 401.7799} C_DIS
LIN {X 87.5257,Y 93.9264,Z 146,A 43.1889,B 23.2866,C -1.3339,E1 23.4327,E2 403.689} C_DIS
LIN {X 90.7178,Y 90.8477,Z 146,A 41.407,B 23.2864,C -1.3392,E1 23.4362,E2 405.4496} C_DIS
LIN {X 93.5361,Y 87.9427,Z 146,A 39.2948,B 23.2874,C -1.3204,E1 23.4404,E2 407.599} C_DIS
LIN {X 96.9473,Y 84.1679,Z 146,A 37.1588,B 23.2873,C -1.3217,E1 23.4443,E2 409.7215} C_DIS
LIN {X 99.6999,Y 80.8887,Z 146,A 35.3864,B 23.2872,C -1.3238,E1 23.4475,E2 411.4797} C_DIS
LIN {X 101.6018,Y 78.4858,Z 146,A 33.8976,B 23.2877,C -1.3146,E1 23.45,E2 412.9841} C_DIS
LIN {X 104.2119,Y 74.9863,Z 146,A 31.9849,B 23.2878,C -1.3115,E1 23.4532,E2 414.8947} C_DIS
LIN {X 106.5545,Y 71.6185,Z 146,A 30.0798,B 23.2883,C -1.3032,E1 23.4562,E2 416.8106} C_DIS
LIN {X 108.2066,Y 69.096,Z 146,A 28.5767,B 23.2889,C -1.292,E1 23.4585,E2 418.3336} C_DIS
LIN {X 109.9041,Y 66.3628,Z 146,A 27.5189,B 23.2881,C -1.3066,E1 23.46,E2 419.349} C_DIS
LIN {X 112.2442,Y 62.3232,Z 146,A 25.2869,B 23.2888,C -1.2936,E1 23.4631,E2 421.601} C_DIS
LIN {X 114.2771,Y 58.5086,Z 146,A 23.4519,B 23.2888,C -1.2929,E1 23.4655,E2 423.4274} C_DIS
LIN {X 115.6072,Y 55.8364,Z 146,A 22.178,B 23.2888,C -1.292,E1 23.467,E2 424.6962} C_DIS
LIN {X 117.2634,Y 52.2662,Z 146,A 19.7006,B 23.2909,C -1.2518,E1 23.47,E2 427.2601} C_DIS
LIN {X 119.3104,Y 47.4117,Z 146,A 17.9744,B 23.2897,C -1.2753,E1 23.4717,E2 428.9169} C_DIS
LIN {X 120.6968,Y 43.7582,Z 146,A 16.3367,B 23.2897,C -1.2753,E1 23.4733,E2 430.5445} C_DIS
LIN {X 122.5151,Y 38.38,Z 146,A 13.6688,B 23.2905,C -1.2611,E1 23.4756,E2 433.2319} C_DIS
LIN {X 123.6336,Y 34.6006,Z 146,A 12.0752,B 23.2903,C -1.2639,E1 23.4769,E2 434.8087} C_DIS
LIN {X 124.5167,Y 31.2756,Z 146,A 10.4433,B 23.2908,C -1.2544,E1 23.478,E2 436.4544} C_DIS
LIN {X 125.4494,Y 27.2946,Z 146,A 8.7254,B 23.2908,C -1.254,E1 23.4791,E2 438.1625} C_DIS
LIN {X 126.0975,Y 24.1233,Z 146,A 7.2965,B 23.291,C -1.2502,E1 23.4798,E2 439.5918} C_DIS
LIN {X 126.6394,Y 21.0947,Z 146,A 5.9181,B 23.2913,C -1.2456,E1 23.4805,E2 440.9731} C_DIS
LIN {X 127.368,Y 16.1317,Z 146,A 3.6783,B 23.2916,C -1.2384,E1 23.4814,E2 443.2166} C_DIS
LIN {X 127.7,Y 13.2473,Z 146,A 1.7165,B 23.2934,C -1.2015,E1 23.482,E2 445.2586} C_DIS
LIN {X 128.1313,Y 8.0597,Z 146,A 0.3849,B 23.2914,C -1.2429,E1 23.4822,E2 446.4777} C_DIS
LIN {X 128.3726,Y 1.7818,Z 146,A -2.5656,B 23.2922,C -1.2265,E1 23.4825,E2 449.4505} C_DIS
LIN {X 128.2959,Y -4.7725,Z 146,A -6.1589,B 23.2943,C -1.184,E1 23.4822,E2 453.1275} C_DIS
LIN {X 128.04,Y -9.3974,Z 146,A -7.6576,B 23.2933,C -1.2053,E1 23.482,E2 454.5629} C_DIS
LIN {X 127.8149,Y -12.0797,Z 146,A -9.1476,B 23.2941,C -1.1871,E1 23.4816,E2 456.0891} C_DIS
LIN {X 127.4555,Y -15.4167,Z 146,A -10.4374,B 23.2939,C -1.1925,E1 23.4812,E2 457.3571} C_DIS
LIN {X 126.8922,Y -19.5167,Z 146,A -12.1045,B 23.2937,C -1.1955,E1 23.4805,E2 459.0061} C_DIS
LIN {X 126.3669,Y -22.6699,Z 146,A -13.5854,B 23.2941,C -1.1882,E1 23.4798,E2 460.4961} C_DIS
LIN {X 125.6553,Y -26.3404,Z 146,A -15.3037,B 23.2945,C -1.1803,E1 23.4788,E2 462.2233} C_DIS
LIN {X 124.8065,Y -30.0967,Z 146,A -16.9066,B 23.2945,C -1.1806,E1 23.4778,E2 463.8155} C_DIS
LIN {X 123.8848,Y -33.6963,Z 146,A -18.6723,B 23.295,C -1.1699,E1 23.4766,E2 465.5969} C_DIS
LIN {X 122.4664,Y -38.5325,Z 146,A -20.8296,B 23.295,C -1.1674,E1 23.4748,E2 467.7473} C_DIS
LIN {X 120.2259,Y -45.0354,Z 146,A -23.8248,B 23.2954,C -1.1615,E1 23.4721,E2 470.7392} C_DIS
LIN {X 118.9893,Y -48.2084,Z 146,A -26.1636,B 23.2974,C -1.1165,E1 23.4695,E2 473.1771} C_DIS
LIN {X 116.6969,Y -53.5204,Z 146,A -27.9326,B 23.296,C -1.1485,E1 23.4676,E2 474.8552} C_DIS
LIN {X 115.2666,Y -56.5341,Z 146,A -29.4003,B 23.2961,C -1.1451,E1 23.4658,E2 476.323} C_DIS
LIN {X 113.8032,Y -59.425,Z 146,A -30.8271,B 23.2963,C -1.1417,E1 23.464,E2 477.7501} C_DIS
LIN {X 112.0192,Y -62.7268,Z 146,A -32.559,B 23.2966,C -1.134,E1 23.4616,E2 479.4918} C_DIS
LIN {X 109.8913,Y -66.384,Z 146,A -35.0146,B 23.2982,C -1.1007,E1 23.458,E2 482.0174} C_DIS
LIN {X 107.2672,Y -70.5455,Z 146,A -36.3878,B 23.2966,C -1.1348,E1 23.4561,E2 483.2974} C_DIS
LIN {X 104.1122,Y -75.1242,Z 146,A -39.1391,B 23.2975,C -1.1146,E1 23.4516,E2 486.085} C_DIS
LIN {X 101.6089,Y -78.4767,Z 146,A -41.2803,B 23.2984,C -1.0961,E1 23.4479,E2 488.2616} C_DIS
LIN {X 99.2943,Y -81.3854,Z 146,A -42.7582,B 23.2982,C -1.1006,E1 23.4453,E2 489.7209} C_DIS
LIN {X 95.9875,Y -85.2608,Z 146,A -44.8658,B 23.2981,C -1.1028,E1 23.4415,E2 491.8126} C_DIS
LIN {X 93.1653,Y -88.3359,Z 146,A -46.4855,B 23.2977,C -1.11,E1 23.4385,E2 493.4064} C_DIS
LIN {X 90.8351,Y -90.7305,Z 146,A -48.2619,B 23.2985,C -1.0924,E1 23.4349,E2 495.2191} C_DIS
LIN {X 86.4459,Y -94.9214,Z 146,A -50.9182,B 23.2987,C -1.0885,E1 23.4295,E2 497.8734} C_DIS
LIN {X 83.4447,Y -97.5707,Z 146,A -52.7649,B 23.299,C -1.0815,E1 23.4256,E2 499.7299} C_DIS
LIN {X 78.6985,Y -101.437,Z 146,A -55.3885,B 23.299,C -1.0807,E1 23.4199,E2 502.3446} C_DIS
LIN {X 75.1546,Y -104.0901,Z 146,A -57.337,B 23.2992,C -1.0779,E1 23.4155,E2 504.2928} C_DIS
LIN {X 72.654,Y -105.8504,Z 146,A -58.7711,B 23.2994,C -1.0718,E1 23.4122,E2 505.737} C_DIS
LIN {X 69.0843,Y -108.2141,Z 146,A -60.6546,B 23.2995,C -1.0694,E1 23.4078,E2 507.6199} C_DIS
LIN {X 65.0004,Y -110.7153,Z 146,A -62.9894,B 23.3001,C -1.0559,E1 23.4021,E2 509.9808} C_DIS
LIN {X 62.1344,Y -112.3486,Z 146,A -64.6393,B 23.3006,C -1.0448,E1 23.398,E2 511.6535} C_DIS
LIN {X 58.4819,Y -114.2907,Z 146,A -65.977,B 23.2997,C -1.0661,E1 23.3949,E2 512.9335} C_DIS
LIN {X 55.4048,Y -115.8134,Z 146,A -67.5063,B 23.2997,C -1.0638,E1 23.391,E2 514.4643} C_DIS
LIN {X 48.6776,Y -118.8001,Z 146,A -70.8838,B 23.3002,C -1.0544,E1 23.3824,E2 517.8566} C_DIS
LIN {X 45.2334,Y -120.1517,Z 146,A -72.4353,B 23.3001,C -1.0569,E1 23.3783,E2 519.3981} C_DIS
LIN {X 42.0909,Y -121.2881,Z 146,A -74.4293,B 23.3012,C -1.0311,E1 23.3729,E2 521.4529} C_DIS
LIN {X 37.9553,Y -122.6459,Z 146,A -75.871,B 23.3003,C -1.0525,E1 23.3692,E2 522.8376} C_DIS
LIN {X 34.6497,Y -123.6199,Z 146,A -77.3839,B 23.3003,C -1.052,E1 23.3652,E2 524.349} C_DIS
LIN {X 31.1082,Y -124.5592,Z 146,A -79.0657,B 23.3004,C -1.0481,E1 23.3606,E2 526.0378} C_DIS
LIN {X 27.2886,Y -125.4506,Z 146,A -80.7068,B 23.3003,C -1.0517,E1 23.3562,E2 527.6676} C_DIS
LIN {X 24.0554,Y -126.1104,Z 146,A -82.1397,B 23.3003,C -1.0523,E1 23.3522,E2 529.097} C_DIS
LIN {X 21.2957,Y -126.6058,Z 146,A -83.5418,B 23.3006,C -1.0443,E1 23.3483,E2 530.5179} C_DIS
LIN {X 15.8327,Y -127.4058,Z 146,A -86.634,B 23.3019,C -1.0133,E1 23.3396,E2 533.6854} C_DIS
LIN {X 10.747,Y -127.9338,Z 146,A -87.9734,B 23.3001,C -1.0561,E1 23.3362,E2 534.9157} C_DIS
LIN {X 4.3092,Y -128.314,Z 146,A -91.0587,B 23.3006,C -1.0452,E1 23.3275,E2 538.0275} C_DIS
LIN {X 0.9203,Y -128.358,Z 146,A -92.4455,B 23.3003,C -1.051,E1 23.3237,E2 539.3994} C_DIS
Enddeposition()
LIN {X 0.9203,Y -128.358,Z 146,A -92.4455,B 23.3003,C -1.051,E1 23.3237,E2 539.3994} C_DIS
Startdeposition()
$VEL.CP = VEL_PRINT
LIN {X 3.8681,Y -127.3692,Z 146,A -90.4349,B 22.4034,C -0.9323,E1 22.4277,E2 537.5831} C_DIS
LIN {X 9.9181,Y -127.0425,Z 146,A -87.6752,B 22.4033,C -0.9349,E1 22.4355,E2 534.8177} C_DIS
LIN {X 12.8831,Y -126.7764,Z 146,A -86.0805,B 22.4028,C -0.9472,E1 22.44,E2 533.1919} C_DIS
LIN {X 16.687,Y -126.3301,Z 146,A -84.0532,B 22.4022,C -0.9623,E1 22.4457,E2 531.127} C_DIS
LIN {X 20.8443,Y -125.711,Z 146,A -82.959,B 22.4036,C -0.9273,E1 22.4485,E2 530.1257} C_DIS
LIN {X 24.1907,Y -125.1103,Z 146,A -81.1704,B 22.403,C -0.9403,E1 22.4535,E2 528.3052} C_DIS
LIN {X 28.0172,Y -124.3096,Z 146,A -79.3282,B 22.4028,C -0.9458,E1 22.4585,E2 526.4516} C_DIS
LIN {X 31.3743,Y -123.5044,Z 146,A -77.8484,B 22.4028,C -0.944,E1 22.4625,E2 524.9789} C_DIS
LIN {X 34.5222,Y -122.6619,Z 146,A -76.3836,B 22.4028,C -0.9455,E1 22.4664,E2 523.5128} C_DIS
LIN {X 38.3444,Y -121.5219,Z 146,A -74.1163,B 22.4019,C -0.9694,E1 22.4727,E2 521.1875} C_DIS
LIN {X 42.2075,Y -120.2349,Z 146,A -72.5536,B 22.4023,C -0.9593,E1 22.4767,E2 519.655} C_DIS
LIN {X 45.9511,Y -118.8537,Z 146,A -70.5225,B 22.4017,C -0.9727,E1 22.4821,E2 517.5937} C_DIS
LIN {X 49.7071,Y -117.334,Z 146,A -68.7749,B 22.4017,C -0.9719,E1 22.4865,E2 515.8529} C_DIS
LIN {X 52.9882,Y -115.8887,Z 146,A -67.6763,B 22.4026,C -0.9504,E1 22.4892,E2 514.8135} C_DIS
LIN {X 55.0878,Y -114.9043,Z 146,A -66.519,B 22.4024,C -0.9574,E1 22.4921,E2 513.6414} C_DIS
LIN {X 58.5523,Y -113.1807,Z 146,A -64.0804,B 22.4009,C -0.9929,E1 22.4984,E2 511.1174} C_DIS
LIN {X 63.1047,Y -110.7065,Z 146,A -62.5639,B 22.4023,C -0.9589,E1 22.5019,E2 509.695} C_DIS
LIN {X 66.0978,Y -108.946,Z 146,A -60.8123,B 22.4018,C -0.9706,E1 22.5061,E2 507.9189} C_DIS
LIN {X 69.6548,Y -106.7072,Z 146,A -58.9247,B 22.4017,C -0.9741,E1 22.5106,E2 506.0291} C_DIS
LIN {X 72.6715,Y -104.6753,Z 146,A -57.342,B 22.4017,C -0.9749,E1 22.5142,E2 504.4504} C_DIS
LIN {X 74.9668,Y -103.0444,Z 146,A -56.0618,B 22.4015,C -0.9782,E1 22.5171,E2 503.1667} C_DIS
LIN {X 80.8537,Y -98.493,Z 146,A -52.3437,B 22.4005,C -1.003,E1 22.5254,E2 499.3996} C_DIS
LIN {X 83.9109,Y -95.9015,Z 146,A -50.9308,B 22.4011,C -0.9886,E1 22.5282,E2 498.0304} C_DIS
LIN {X 87.5083,Y -92.6304,Z 146,A -48.4425,B 22.4002,C -1.008,E1 22.5334,E2 495.5029} C_DIS
LIN {X 90.1774,Y -90.0347,Z 146,A -46.7016,B 22.3999,C -1.0153,E1 22.5369,E2 493.7514} C_DIS
LIN {X 93.0135,Y -87.1018,Z 146,A -45.2682,B 22.4006,C -1.0007,E1 22.5395,E2 492.3631} C_DIS
LIN {X 95.8649,Y -83.9529,Z 146,A -42.936,B 22.3995,C -1.0257,E1 22.5439,E2 489.9774} C_DIS
LIN {X 98.6281,Y -80.6884,Z 146,A -40.7473,B 22.3987,C -1.0435,E1 22.5478,E2 487.7538} C_DIS
LIN {X 102.1255,Y -76.2136,Z 146,A -39.2886,B 22.4007,C -0.998,E1 22.5501,E2 486.4217} C_DIS
LIN {X 105.8977,Y -70.8789,Z 146,A -36.0965,B 22.3998,C -1.0181,E1 22.5553,E2 483.1947} C_DIS
LIN {X 108.8821,Y -66.2034,Z 146,A -33.8231,B 22.4,C -1.0146,E1 22.5586,E2 480.9433} C_DIS
LIN {X 110.1489,Y -64.0735,Z 146,A -32.3947,B 22.3992,C -1.0328,E1 22.5607,E2 479.4758} C_DIS
LIN {X 112.1951,Y -60.4185,Z 146,A -30.6021,B 22.3992,C -1.034,E1 22.5631,E2 477.6908} C_DIS
LIN {X 113.6111,Y -57.7076,Z 146,A -29.2756,B 22.399,C -1.0357,E1 22.5648,E2 476.3677} C_DIS
LIN {X 115.0803,Y -54.7194,Z 146,A -27.7387,B 22.3988,C -1.0421,E1 22.5667,E2 474.8235} C_DIS
LIN {X 118.5536,Y -46.7232,Z 146,A -23.9861,B 22.3986,C -1.0459,E1 22.5708,E2 471.0843} C_DIS
LIN {X 121.0787,Y -39.7231,Z 146,A -20.676,B 22.3982,C -1.0544,E1 22.5739,E2 467.7728} C_DIS
LIN {X 122.1742,Y -36.212,Z 146,A -19.0129,B 22.398,C -1.0601,E1 22.5752,E2 466.1057} C_DIS
LIN {X 122.7899,Y -34.0645,Z 146,A -17.905,B 22.3976,C -1.0682,E1 22.5761,E2 464.9838} C_DIS
LIN {X 123.8415,Y -30.0166,Z 146,A -16.0335,B 22.3973,C -1.0737,E1 22.5773,E2 463.1101} C_DIS
LIN {X 124.7187,Y -26.144,Z 146,A -14.1309,B 22.3968,C -1.085,E1 22.5785,E2 461.1906} C_DIS
LIN {X 125.4522,Y -22.3489,Z 146,A -12.4932,B 22.3968,C -1.0857,E1 22.5793,E2 459.5618} C_DIS
LIN {X 126.1403,Y -18.0653,Z 146,A -9.9842,B 22.3952,C -1.1189,E1 22.5803,E2 456.9829} C_DIS
LIN {X 126.7471,Y -13.1584,Z 146,A -8.2958,B 22.3961,C -1.1002,E1 22.5808,E2 455.3546} C_DIS
LIN {X 127.1205,Y -8.8502,Z 146,A -6.5402,B 22.3963,C -1.0974,E1 22.5812,E2 453.618} C_DIS
LIN {X 127.3619,Y -4.129,Z 146,A -3.946,B 22.3949,C -1.1268,E1 22.5815,E2 450.9647} C_DIS
LIN {X 127.4319,Y -0.0791,Z 146,A -2.6625,B 22.3958,C -1.1067,E1 22.5815,E2 449.7421} C_DIS
LIN {X 127.2231,Y 7.2381,Z 146,A 0.7437,B 22.3951,C -1.1228,E1 22.5812,E2 446.317} C_DIS
LIN {X 126.8282,Y 12.3442,Z 146,A 2.8235,B 22.3952,C -1.1195,E1 22.5807,E2 444.2597} C_DIS
LIN {X 126.5442,Y 14.9771,Z 146,A 4.1607,B 22.3947,C -1.1302,E1 22.5803,E2 442.9033} C_DIS
LIN {X 126.1375,Y 18.0845,Z 146,A 5.8697,B 22.3938,C -1.1491,E1 22.5796,E2 441.1567} C_DIS
LIN {X 125.6354,Y 21.2971,Z 146,A 6.9408,B 22.3945,C -1.1349,E1 22.5792,E2 440.1295} C_DIS
LIN {X 125.1091,Y 24.1971,Z 146,A 8.36,B 22.3941,C -1.1435,E1 22.5784,E2 438.6972} C_DIS
LIN {X 124.2697,Y 28.1916,Z 146,A 10.1399,B 22.3939,C -1.1466,E1 22.5774,E2 436.9211} C_DIS
LIN {X 123.5225,Y 31.3033,Z 146,A 11.5774,B 22.3937,C -1.1509,E1 22.5764,E2 435.4816} C_DIS
LIN {X 122.6236,Y 34.6591,Z 146,A 13.1466,B 22.3935,C -1.156,E1 22.5752,E2 433.9093} C_DIS
LIN {X 121.5611,Y 38.2217,Z 146,A 15.2203,B 22.3923,C -1.1803,E1 22.5735,E2 431.7857} C_DIS
LIN {X 120.3858,Y 41.7722,Z 146,A 16.5191,B 22.3929,C -1.167,E1 22.5723,E2 430.5298} C_DIS
LIN {X 118.439,Y 47.0139,Z 146,A 19.6745,B 22.391,C -1.205,E1 22.5691,E2 427.295} C_DIS
LIN {X 116.4242,Y 51.7988,Z 146,A 21.0411,B 22.393,C -1.1656,E1 22.5677,E2 426.0397} C_DIS
LIN {X 114.9145,Y 55.0664,Z 146,A 22.922,B 22.3921,C -1.1826,E1 22.5654,E2 424.1259} C_DIS
LIN {X 113.4517,Y 58.0206,Z 146,A 24.3916,B 22.392,C -1.1861,E1 22.5635,E2 422.656} C_DIS
LIN {X 111.5231,Y 61.6501,Z 146,A 26.5784,B 22.3909,C -1.2072,E1 22.5606,E2 420.4271} C_DIS
LIN {X 109.7228,Y 64.8007,Z 146,A 27.665,B 22.392,C -1.1858,E1 22.5591,E2 419.4026} C_DIS
LIN {X 107.4402,Y 68.5184,Z 146,A 29.669,B 22.3916,C -1.1929,E1 22.5562,E2 417.3915} C_DIS
LIN {X 105.6184,Y 71.2945,Z 146,A 31.319,B 22.3911,C -1.2041,E1 22.5536,E2 415.7215} C_DIS
LIN {X 103.3617,Y 74.529,Z 146,A 33.1345,B 22.3907,C -1.2106,E1 22.5506,E2 413.8991} C_DIS
LIN {X 100.4516,Y 78.4074,Z 146,A 34.9945,B 22.3912,C -1.2009,E1 22.5475,E2 412.0745} C_DIS
LIN {X 98.5927,Y 80.7317,Z 146,A 36.6007,B 22.3904,C -1.2166,E1 22.5447,E2 410.4356} C_DIS
LIN {X 95.7228,Y 84.1154,Z 146,A 38.6304,B 22.3901,C -1.2228,E1 22.5409,E2 408.4} C_DIS
LIN {X 91.6081,Y 88.5781,Z 146,A 40.9944,B 22.3907,C -1.2119,E1 22.5365,E2 406.0763} C_DIS
LIN {X 89.7193,Y 90.4908,Z 146,A 42.5088,B 22.3898,C -1.2287,E1 22.5335,E2 404.5253} C_DIS
LIN {X 86.5225,Y 93.5528,Z 146,A 44.3309,B 22.39,C -1.225,E1 22.5298,E2 402.7213} C_DIS
LIN {X 84.0533,Y 95.7773,Z 146,A 45.9821,B 22.3894,C -1.2352,E1 22.5263,E2 401.0507} C_DIS
LIN {X 80.6497,Y 98.6597,Z 146,A 47.8752,B 22.3895,C -1.2339,E1 22.5223,E2 399.1694} C_DIS
LIN {X 77.6475,Y 101.04,Z 146,A 49.7131,B 22.3891,C -1.2424,E1 22.5182,E2 397.317} C_DIS
LIN {X 73.9816,Y 103.7539,Z 146,A 51.7506,B 22.3889,C -1.2453,E1 22.5136,E2 395.2799} C_DIS
LIN {X 70.3364,Y 106.2591,Z 146,A 53.6959,B 22.3889,C -1.2466,E1 22.5091,E2 393.3387} C_DIS
LIN {X 66.8183,Y 108.5057,Z 146,A 55.6971,B 22.3884,C -1.2552,E1 22.5043,E2 391.3221} C_DIS
LIN {X 62.0123,Y 111.3225,Z 146,A 57.9243,B 22.3889,C -1.2461,E1 22.499,E2 389.1262} C_DIS
LIN {X 59.0732,Y 112.9071,Z 146,A 59.4707,B 22.3887,C -1.2503,E1 22.4952,E2 387.574} C_DIS
LIN {X 56.0471,Y 114.4399,Z 146,A 61.0881,B 22.3883,C -1.2564,E1 22.4911,E2 385.9455} C_DIS
LIN {X 52.3304,Y 116.1864,Z 146,A 62.8584,B 22.3883,C -1.2551,E1 22.4866,E2 384.1836} C_DIS
LIN {X 49.0424,Y 117.6116,Z 146,A 64.4114,B 22.3884,C -1.2543,E1 22.4827,E2 382.6371} C_DIS
LIN {X 45.0128,Y 119.2125,Z 146,A 66.5373,B 22.3879,C -1.2642,E1 22.4771,E2 380.4905} C_DIS
LIN {X 40.3233,Y 120.8789,Z 146,A 68.8221,B 22.3877,C -1.2683,E1 22.471,E2 378.2001} C_DIS
LIN {X 36.0258,Y 122.2288,Z 146,A 70.6961,B 22.388,C -1.263,E1 22.4661,E2 376.3436} C_DIS
LIN {X 32.5668,Y 123.1956,Z 146,A 72.3424,B 22.3878,C -1.2655,E1 22.4616,E2 374.6938} C_DIS
LIN {X 28.4109,Y 124.2196,Z 146,A 74.1852,B 22.388,C -1.2629,E1 22.4566,E2 372.8606} C_DIS
LIN {X 24.7406,Y 125.0043,Z 146,A 76.0253,B 22.3876,C -1.2705,E1 22.4516,E2 371.0032} C_DIS
LIN {X 20.8196,Y 125.7151,Z 146,A 77.725,B 22.3878,C -1.2671,E1 22.4469,E2 369.3145} C_DIS
LIN {X 14.0281,Y 126.6535,Z 146,A 80.6798,B 22.388,C -1.2622,E1 22.4388,E2 366.3753} C_DIS
LIN {X 10.7972,Y 126.9692,Z 146,A 82.1664,B 22.388,C -1.2635,E1 22.4346,E2 364.8861} C_DIS
LIN {X 5.9366,Y 127.29,Z 146,A 84.4463,B 22.3877,C -1.2675,E1 22.4282,E2 362.5968} C_DIS
LIN {X -0.1592,Y 127.4286,Z 146,A 87.2375,B 22.3877,C -1.2693,E1 22.4204,E2 359.8013} C_DIS
LIN {X -4.1957,Y 127.3601,Z 146,A 89.0464,B 22.3877,C -1.2686,E1 22.4154,E2 357.9942} C_DIS
LIN {X -8.8027,Y 127.1239,Z 146,A 91.357,B 22.3872,C -1.2782,E1 22.4089,E2 355.6575} C_DIS
LIN {X -12.0542,Y 126.856,Z 146,A 92.465,B 22.388,C -1.2618,E1 22.4059,E2 354.5917} C_DIS
LIN {X -15.3498,Y 126.4997,Z 146,A 94.0423,B 22.3879,C -1.2648,E1 22.4015,E2 353.0055} C_DIS
LIN {X -20.0729,Y 125.8378,Z 146,A 96.0565,B 22.3883,C -1.2578,E1 22.396,E2 351.0079} C_DIS
LIN {X -22.62,Y 125.4037,Z 146,A 97.259,B 22.3883,C -1.2587,E1 22.3927,E2 349.8016} C_DIS
LIN {X -25.8798,Y 124.7725,Z 146,A 98.9065,B 22.3879,C -1.2642,E1 22.3881,E2 348.1376} C_DIS
LIN {X -29.9224,Y 123.8642,Z 146,A 100.6608,B 22.3883,C -1.2579,E1 22.3834,E2 346.3973} C_DIS
LIN {X -33.2862,Y 123.0038,Z 146,A 102.3487,B 22.388,C -1.2618,E1 22.3788,E2 344.6963} C_DIS
LIN {X -41.2412,Y 120.5699,Z 146,A 105.8832,B 22.3887,C -1.2487,E1 22.3695,E2 341.1892} C_DIS
LIN {X -47.0527,Y 118.4234,Z 146,A 108.6865,B 22.3889,C -1.2458,E1 22.3621,E2 338.3869} C_DIS
LIN {X -50.906,Y 116.8176,Z 146,A 110.7614,B 22.3886,C -1.2516,E1 22.3567,E2 336.2915} C_DIS
LIN {X -54.4859,Y 115.1918,Z 146,A 112.2872,B 22.3893,C -1.2386,E1 22.353,E2 334.7954} C_DIS
LIN {X -58.2794,Y 113.32,Z 146,A 114.4127,B 22.3889,C -1.2451,E1 22.3476,E2 332.6466} C_DIS
LIN {X -62.1421,Y 111.2501,Z 146,A 116.4448,B 22.3889,C -1.2443,E1 22.3426,E2 330.6099} C_DIS
LIN {X -66.1157,Y 108.9352,Z 146,A 118.458,B 22.3893,C -1.2383,E1 22.3378,E2 328.6055} C_DIS
LIN {X -69.6455,Y 106.7133,Z 146,A 120.3748,B 22.3893,C -1.2366,E1 22.3333,E2 326.6864} C_DIS
LIN {X -75.4594,Y 102.6839,Z 146,A 123.5704,B 22.3897,C -1.2308,E1 22.326,E2 323.4936} C_DIS
LIN {X -79.0063,Y 99.9813,Z 146,A 125.5401,B 22.39,C -1.2251,E1 22.3217,E2 321.5307} C_DIS
LIN {X -83.0662,Y 96.6341,Z 146,A 128.3135,B 22.3894,C -1.237,E1 22.3157,E2 318.7139} C_DIS
LIN {X -85.9984,Y 94.0345,Z 146,A 129.5955,B 22.3906,C -1.2129,E1 22.3131,E2 317.4895} C_DIS
LIN {X -88.7082,Y 91.4821,Z 146,A 131.5365,B 22.3902,C -1.2201,E1 22.3092,E2 315.5205} C_DIS
LIN {X -92.1122,Y 88.0537,Z 146,A 133.988,B 22.3899,C -1.2265,E1 22.3043,E2 313.0403} C_DIS
LIN {X -94.8765,Y 85.0681,Z 146,A 135.369,B 22.3911,C -1.2033,E1 22.3019,E2 311.7135} C_DIS
LIN {X -97.4663,Y 82.0884,Z 146,A 137.7242,B 22.3901,C -1.2228,E1 22.2975,E2 309.2946} C_DIS
LIN {X -100.3734,Y 78.5071,Z 146,A 139.4743,B 22.3911,C -1.2039,E1 22.2945,E2 307.5852} C_DIS
LIN {X -103.2098,Y 74.7387,Z 146,A 141.3692,B 22.3918,C -1.1889,E1 22.2914,E2 305.7195} C_DIS
LIN {X -105.2452,Y 71.8448,Z 146,A 143.0132,B 22.3919,C -1.1867,E1 22.2888,E2 304.072} C_DIS
LIN {X -107.5577,Y 68.3345,Z 146,A 144.9773,B 22.392,C -1.1845,E1 22.2858,E2 302.1027} C_DIS
LIN {X -109.8442,Y 64.594,Z 146,A 146.9252,B 22.3924,C -1.1779,E1 22.2831,E2 300.1606} C_DIS
LIN {X -112.0063,Y 60.7684,Z 146,A 148.9593,B 22.3925,C -1.1746,E1 22.2803,E2 298.1232} C_DIS
LIN {X -113.7745,Y 57.3866,Z 146,A 150.6656,B 22.3928,C -1.1692,E1 22.2781,E2 296.4208} C_DIS
LIN {X -115.5634,Y 53.6916,Z 146,A 152.8089,B 22.3925,C -1.176,E1 22.2756,E2 294.2466} C_DIS
LIN {X -117.0395,Y 50.3927,Z 146,A 154.0651,B 22.3935,C -1.1559,E1 22.2742,E2 293.0354} C_DIS
LIN {X -118.1787,Y 47.6597,Z 146,A 155.4121,B 22.3936,C -1.1525,E1 22.2728,E2 291.6889} C_DIS
LIN {X -119.465,Y 44.3387,Z 146,A 156.9385,B 22.394,C -1.1446,E1 22.2713,E2 290.1739} C_DIS
LIN {X -120.812,Y 40.524,Z 146,A 158.611,B 22.3946,C -1.133,E1 22.2698,E2 288.5212} C_DIS
LIN {X -121.4979,Y 38.4197,Z 146,A 160.504,B 22.3929,C -1.1666,E1 22.2681,E2 286.527} C_DIS
LIN {X -122.9219,Y 33.5925,Z 146,A 162.0983,B 22.3946,C -1.1321,E1 22.267,E2 285.0136} C_DIS
LIN {X -124.8649,Y 25.4258,Z 146,A 165.898,B 22.3951,C -1.1211,E1 22.2646,E2 281.2177} C_DIS
LIN {X -125.4788,Y 22.2002,Z 146,A 167.4843,B 22.3951,C -1.1209,E1 22.2638,E2 279.6213} C_DIS
LIN {X -126.1301,Y 18.1368,Z 146,A 169.2999,B 22.3955,C -1.1135,E1 22.263,E2 277.8129} C_DIS
LIN {X -126.5836,Y 14.6466,Z 146,A 170.9707,B 22.3955,C -1.1121,E1 22.2624,E2 276.1347} C_DIS
LIN {X -126.9779,Y 10.6937,Z 146,A 172.708,B 22.3959,C -1.1043,E1 22.262,E2 274.406} C_DIS
LIN {X -127.2638,Y 6.456,Z 146,A 174.641,B 22.3962,C -1.0991,E1 22.2617,E2 272.4735} C_DIS
LIN {X -127.4077,Y 2.2517,Z 146,A 176.4804,B 22.3966,C -1.091,E1 22.2615,E2 270.6433} C_DIS
LIN {X -127.4264,Y -0.8044,Z 146,A 177.9705,B 22.3966,C -1.0913,E1 22.2615,E2 269.1422} C_DIS
LIN {X -127.3337,Y -4.8893,Z 146,A 179.7608,B 22.3969,C -1.0835,E1 22.2617,E2 267.3602} C_DIS
LIN {X -127.1092,Y -9.0049,Z 146,A -178.3236,B 22.3971,C -1.0801,E1 22.262,E2 265.4404} C_DIS
LIN {X -126.8215,Y -12.4142,Z 146,A -176.81,B 22.3973,C -1.0742,E1 22.2624,E2 263.9322} C_DIS
LIN {X -126.3602,Y -16.4574,Z 146,A -174.9914,B 22.3976,C -1.068,E1 22.263,E2 262.1177} C_DIS
LIN {X -125.8139,Y -20.2266,Z 146,A -173.1299,B 22.3976,C -1.0687,E1 22.2638,E2 260.2418} C_DIS
LIN {X -125.1417,Y -24.0265,Z 146,A -171.5405,B 22.3981,C -1.0574,E1 22.2646,E2 258.6717} C_DIS
LIN {X -124.4829,Y -27.2368,Z 146,A -170.0049,B 22.3981,C -1.0553,E1 22.2655,E2 257.1312} C_DIS
LIN {X -123.5639,Y -31.14,Z 146,A -167.7922,B 22.3977,C -1.0667,E1 22.267,E2 254.8739} C_DIS
LIN {X -122.5508,Y -34.9193,Z 146,A -166.4989,B 22.3988,C -1.0421,E1 22.268,E2 253.6371} C_DIS
LIN {X -120.7638,Y -40.6687,Z 146,A -163.733,B 22.399,C -1.0364,E1 22.2703,E2 250.8683} C_DIS
LIN {X -119.6151,Y -43.9368,Z 146,A -162.1848,B 22.3992,C -1.0314,E1 22.2718,E2 249.3234} C_DIS
LIN {X -118.785,Y -46.1278,Z 146,A -161.1013,B 22.3993,C -1.0296,E1 22.2729,E2 248.2378} C_DIS
LIN {X -117.5581,Y -49.1705,Z 146,A -159.6426,B 22.3995,C -1.0246,E1 22.2744,E2 246.7829} C_DIS
LIN {X -116.2131,Y -52.2707,Z 146,A -158.0873,B 22.3997,C -1.0218,E1 22.2762,E2 245.2256} C_DIS
LIN {X -114.751,Y -55.4087,Z 146,A -156.5493,B 22.3999,C -1.0166,E1 22.278,E2 243.6917} C_DIS
LIN {X -113.3954,Y -58.1312,Z 146,A -155.075,B 22.3999,C -1.0173,E1 22.2799,E2 242.2067} C_DIS
LIN {X -110.2298,Y -63.9337,Z 146,A -152.2953,B 22.4005,C -1.0012,E1 22.2836,E2 239.453} C_DIS
LIN {X -108.5207,Y -66.7938,Z 146,A -150.5301,B 22.4002,C -1.0083,E1 22.2862,E2 237.6587} C_DIS
LIN {X -106.1914,Y -70.4389,Z 146,A -148.3311,B 22.4,C -1.014,E1 22.2896,E2 235.4323} C_DIS
LIN {X -104.2726,Y -73.2488,Z 146,A -147.2245,B 22.4009,C -0.9924,E1 22.2913,E2 234.3765} C_DIS
LIN {X -102.3554,Y -75.9049,Z 146,A -145.1596,B 22.4,C -1.0136,E1 22.2948,E2 232.2442} C_DIS
LIN {X -99.8175,Y -79.2125,Z 146,A -143.7017,B 22.4009,C -0.9916,E1 22.2973,E2 230.8367} C_DIS
LIN {X -97.1366,Y -82.4779,Z 146,A -141.7703,B 22.4011,C -0.9885,E1 22.3007,E2 228.9035} C_DIS
LIN {X -94.2019,Y -85.8148,Z 146,A -139.796,B 22.4013,C -0.983,E1 22.3044,E2 226.9338} C_DIS
LIN {X -91.396,Y -88.7972,Z 146,A -137.9338,B 22.4014,C -0.9799,E1 22.308,E2 225.0707} C_DIS
LIN {X -88.3222,Y -91.8556,Z 146,A -135.9255,B 22.4014,C -0.9782,E1 22.312,E2 223.0572} C_DIS
LIN {X -85.1167,Y -94.8329,Z 146,A -133.9731,B 22.4017,C -0.9737,E1 22.316,E2 221.1078} C_DIS
LIN {X -81.6674,Y -97.8194,Z 146,A -131.9293,B 22.4019,C -0.9694,E1 22.3204,E2 219.0664} C_DIS
LIN {X -78.893,Y -100.0703,Z 146,A -130.2894,B 22.4019,C -0.9679,E1 22.324,E2 217.4236} C_DIS
LIN {X -74.2201,Y -103.5833,Z 146,A -127.6892,B 22.4022,C -0.9621,E1 22.3298,E2 214.8282} C_DIS
LIN {X -71.1492,Y -105.7167,Z 146,A -125.9588,B 22.4022,C -0.9614,E1 22.3338,E2 213.0931} C_DIS
LIN {X -67.3746,Y -108.1609,Z 146,A -124.1073,B 22.4026,C -0.951,E1 22.3381,E2 211.2624} C_DIS
LIN {X -64.2542,Y -110.0438,Z 146,A -122.4139,B 22.4026,C -0.951,E1 22.3422,E2 209.5633} C_DIS
LIN {X -61.0287,Y -111.8643,Z 146,A -120.636,B 22.4026,C -0.9535,E1 22.3466,E2 207.7728} C_DIS
LIN {X -57.7814,Y -113.5735,Z 146,A -119.0224,B 22.4026,C -0.9498,E1 22.3505,E2 206.1639} C_DIS
LIN {X -54.8138,Y -115.0352,Z 146,A -117.574,B 22.4028,C -0.9463,E1 22.3542,E2 204.7204} C_DIS
LIN {X -51.6752,Y -116.4795,Z 146,A -116.0131,B 22.4028,C -0.9449,E1 22.3582,E2 203.159} C_DIS
LIN {X -47.331,Y -118.3112,Z 146,A -113.9078,B 22.403,C -0.9421,E1 22.3636,E2 201.0558} C_DIS
LIN {X -43.5506,Y -119.7544,Z 146,A -111.7727,B 22.4025,C -0.9542,E1 22.3693,E2 198.8839} C_DIS
LIN {X -39.9104,Y -121.0164,Z 146,A -110.2271,B 22.4029,C -0.9446,E1 22.3733,E2 197.3603} C_DIS
Enddeposition()
END
